TYPE "UDT_PECUpdateStatistics"
TITLE = UDT_PECupdateStatistics
VERSION : 0.1
//User-defined structure of FB_PECUpdate function block statistics.
   STRUCT
      PEC { S7_SetPoint := 'False'} : "UDT_PECStatistics";   // PEC Statistics
      TooManyLost { S7_SetPoint := 'False'} : "UDT_EventStatistic";   // Too many lost parcels
      TotalNrOfParcels : DInt;   // Total number of parcels
   END_STRUCT;

END_TYPE

TYPE "UDT_UnknownGIN"
TITLE = UDT_UnknownGIN
VERSION : 0.1
//User-defined structure of unknown GIN range.
   STRUCT
      Start : Int := 1;   // Unknown GIN range start value
      End : Int := 199;   // Unknown GIN range end value
      GIN : Int := 0;   // Las generated unknown GIN
   END_STRUCT;

END_TYPE

TYPE "UDT_AixPlcFullIn"
VERSION : 0.1
   STRUCT
      ConveyStopStatus { ExternalVisible := 'False'} : Struct   // Status of ConveyStop
         Bit08 { ExternalAccessible := 'False'; ExternalVisible := 'False'; ExternalWritable := 'False'} : Bool;   // Reserved
         Bit09 { ExternalAccessible := 'False'; ExternalVisible := 'False'; ExternalWritable := 'False'} : Bool;   // Reserved
         StopActiveCommandPLC { ExternalAccessible := 'False'; ExternalVisible := 'False'; ExternalWritable := 'False'} : Bool;   // Stop active due to stop command from the PLC
         Bit11 { ExternalAccessible := 'False'; ExternalVisible := 'False'; ExternalWritable := 'False'} : Bool;   // Reserved
         Bit12 { ExternalAccessible := 'False'; ExternalVisible := 'False'; ExternalWritable := 'False'} : Bool;   // Reserved
         Bit13 { ExternalAccessible := 'False'; ExternalVisible := 'False'; ExternalWritable := 'False'} : Bool;   // Reserved
         Bit14 { ExternalAccessible := 'False'; ExternalVisible := 'False'; ExternalWritable := 'False'} : Bool;   // Reserved
         Bit15 { ExternalAccessible := 'False'; ExternalVisible := 'False'; ExternalWritable := 'False'} : Bool;   // Reserved
         Bit00 { ExternalAccessible := 'False'; ExternalVisible := 'False'; ExternalWritable := 'False'} : Bool;   // Reserved
         Bit01 { ExternalAccessible := 'False'; ExternalVisible := 'False'; ExternalWritable := 'False'} : Bool;   // Reserved
         Bit02 { ExternalAccessible := 'False'; ExternalVisible := 'False'; ExternalWritable := 'False'} : Bool;   // Reserved
         Bit03 { ExternalAccessible := 'False'; ExternalVisible := 'False'; ExternalWritable := 'False'} : Bool;   // Reserved
         Bit04 { ExternalAccessible := 'False'; ExternalVisible := 'False'; ExternalWritable := 'False'} : Bool;   // Reserved
         StopActiveOtherModule { ExternalAccessible := 'False'; ExternalVisible := 'False'; ExternalWritable := 'False'} : Bool;   // Stop condition is active on a module in the ConveyStop group
         StopActiveLostConn { ExternalAccessible := 'False'; ExternalVisible := 'False'; ExternalWritable := 'False'} : Bool;   // Stop is active due to a loss of communication connection
         StopActiveLostPLC { ExternalAccessible := 'False'; ExternalVisible := 'False'; ExternalWritable := 'False'} : Bool;   // Stop active due to a loss of connection with the PLC
      END_STRUCT;
      AllSensorPortInputs { ExternalVisible := 'False'} : Struct   // Left and Right Sensor Port inputs
         Bit08 { ExternalAccessible := 'False'; ExternalVisible := 'False'; ExternalWritable := 'False'} : Bool;   // Reserved
         Bit09 { ExternalAccessible := 'False'; ExternalVisible := 'False'; ExternalWritable := 'False'} : Bool;   // Reserved
         Bit10 { ExternalAccessible := 'False'; ExternalVisible := 'False'; ExternalWritable := 'False'} : Bool;   // Reserved
         Bit11 { ExternalAccessible := 'False'; ExternalVisible := 'False'; ExternalWritable := 'False'} : Bool;   // Reserved
         Bit12 { ExternalAccessible := 'False'; ExternalVisible := 'False'; ExternalWritable := 'False'} : Bool;   // Reserved
         Bit13 { ExternalAccessible := 'False'; ExternalVisible := 'False'; ExternalWritable := 'False'} : Bool;   // Reserved
         Bit14 { ExternalAccessible := 'False'; ExternalVisible := 'False'; ExternalWritable := 'False'} : Bool;   // Reserved
         Heartbeat { ExternalAccessible := 'False'; ExternalVisible := 'False'; ExternalWritable := 'False'} : Bool;   // This bit toggles every 2 seconds
         LeftPin2 { ExternalAccessible := 'False'; ExternalVisible := 'False'; ExternalWritable := 'False'} : Bool;   // Left sensor port Pin2 state
         Bit01 { ExternalAccessible := 'False'; ExternalVisible := 'False'; ExternalWritable := 'False'} : Bool;   // Reserved
         RightPin2 { ExternalAccessible := 'False'; ExternalVisible := 'False'; ExternalWritable := 'False'} : Bool;   // Right sensor port Pin2 state
         Bit03 { ExternalAccessible := 'False'; ExternalVisible := 'False'; ExternalWritable := 'False'} : Bool;   // Reserved
         LeftSensor { ExternalAccessible := 'False'; ExternalVisible := 'False'; ExternalWritable := 'False'} : Bool;   // Left sensor port Pin4 state
         Bit05 { ExternalAccessible := 'False'; ExternalVisible := 'False'; ExternalWritable := 'False'} : Bool;   // Reserved
         RightSensor { ExternalAccessible := 'False'; ExternalVisible := 'False'; ExternalWritable := 'False'} : Bool;   // Right sensor port Pin4 state
         Bit07 { ExternalAccessible := 'False'; ExternalVisible := 'False'; ExternalWritable := 'False'} : Bool;   // Reserved
      END_STRUCT;
      SensorDetect { ExternalVisible := 'False'} : Struct   // Sensor detection
         Bits08_15 { ExternalVisible := 'False'} : SInt;   // Reserved
         RightSensorDetect { ExternalAccessible := 'False'; ExternalVisible := 'False'; ExternalWritable := 'False'} : Bool;   // True when sensor is detected
         LeftSensorDetect { ExternalAccessible := 'False'; ExternalVisible := 'False'; ExternalWritable := 'False'} : Bool;   // True when sensor is detected
         Bit02 { ExternalAccessible := 'False'; ExternalVisible := 'False'; ExternalWritable := 'False'} : Bool;   // Reserved
         Bit03 { ExternalAccessible := 'False'; ExternalVisible := 'False'; ExternalWritable := 'False'} : Bool;   // Reserved
         Bit04 { ExternalAccessible := 'False'; ExternalVisible := 'False'; ExternalWritable := 'False'} : Bool;   // Reserved
         Bit05 { ExternalAccessible := 'False'; ExternalVisible := 'False'; ExternalWritable := 'False'} : Bool;   // Reserved
         Bit06 { ExternalAccessible := 'False'; ExternalVisible := 'False'; ExternalWritable := 'False'} : Bool;   // Reserved
         Bit07 { ExternalAccessible := 'False'; ExternalVisible := 'False'; ExternalWritable := 'False'} : Bool;   // Reserved
      END_STRUCT;
      VoltageMotors { ExternalVisible := 'False'} : Int;   // The Voltage applied to the module's motor power connection in millivolts
      LeftMotorCurrent { ExternalVisible := 'False'} : Int;   // Left motor running current in milliamperes
      LeftMotorFreq { ExternalVisible := 'False'} : Int;   // Left motor running electrical frequency in Hz
      LeftMotorCalcTemp { ExternalVisible := 'False'} : Byte;   // Left motor temperature in degrees C
      ModuleTemp { ExternalVisible := 'False'} : Byte;   // Module CPU temperature in degrees C
      LeftMotorDiagnostic { ExternalVisible := 'False'} : Struct   // Left motor diagnostics .
         Overheat { ExternalAccessible := 'False'; ExternalVisible := 'False'; ExternalWritable := 'False'} : Bool;   // Left motor temperature has exceeded 105 degrees Celsius
         MaxTorque { ExternalAccessible := 'False'; ExternalVisible := 'False'; ExternalWritable := 'False'} : Bool;   // Left motor at maximum torque output
         ShortCircuit { ExternalAccessible := 'False'; ExternalVisible := 'False'; ExternalWritable := 'False'} : Bool;   // Left motor short circuit
         MotorNotConnected { ExternalAccessible := 'False'; ExternalVisible := 'False'; ExternalWritable := 'False'} : Bool;   // Left motor is not connected
         Overload { ExternalAccessible := 'False'; ExternalVisible := 'False'; ExternalWritable := 'False'} : Bool;   // Left motor overloaded after more than 20 seconds in Stalled
         Stalled { ExternalAccessible := 'False'; ExternalVisible := 'False'; ExternalWritable := 'False'} : Bool;   // Left motor stalled and speed is less than 10% of the set speed
         BadHall { ExternalAccessible := 'False'; ExternalVisible := 'False'; ExternalWritable := 'False'} : Bool;   // Left motor Hall Effect Sensor error active
         MotorNotUsed { ExternalAccessible := 'False'; ExternalVisible := 'False'; ExternalWritable := 'False'} : Bool;   // Left motor not used
         MotorStatus1 { ExternalAccessible := 'False'; ExternalVisible := 'False'; ExternalWritable := 'False'} : Bool;   // Left motor running and direction status
         MotorStatus2 { ExternalAccessible := 'False'; ExternalVisible := 'False'; ExternalWritable := 'False'} : Bool;   // Left motor running and direction status
         MotorPortinDOmode { ExternalAccessible := 'False'; ExternalVisible := 'False'; ExternalWritable := 'False'} : Bool;   // Left motor port is in digital Output mode .
         ReservedBit03 { ExternalAccessible := 'False'; ExternalVisible := 'False'; ExternalWritable := 'False'} : Bool;   // Reserved
         ReservedBit04 { ExternalAccessible := 'False'; ExternalVisible := 'False'; ExternalWritable := 'False'} : Bool;   // Reserved
         BoardOverheat { ExternalAccessible := 'False'; ExternalVisible := 'False'; ExternalWritable := 'False'} : Bool;   // Board temperature has exceeded 90 degrees Celsius
         OverVoltage { ExternalAccessible := 'False'; ExternalVisible := 'False'; ExternalWritable := 'False'} : Bool;   // Supply voltage + motor back EMF exceeded 30 volts
         LowVoltage { ExternalAccessible := 'False'; ExternalVisible := 'False'; ExternalWritable := 'False'} : Bool;   // Module power supply is less than 18 Volts
      END_STRUCT;
      RightMotorCurrent { ExternalVisible := 'False'} : Int;   // Right motor running current in milliamperes
      RightMotorFreq { ExternalVisible := 'False'} : Int;   // Right motor running electrical frequency in Hz
      RightMotorCalcTemp { ExternalVisible := 'False'} : Byte;   // Right motor temperature in degrees Celsius
      ModuleTemp1 { ExternalVisible := 'False'} : Byte;   // Module PCB temperature in degrees C (same as ModuleTemp tag)
      RightMotorDiagnostic { ExternalVisible := 'False'} : Struct   // Right motor diagnostics .
         Overheat { ExternalAccessible := 'False'; ExternalVisible := 'False'; ExternalWritable := 'False'} : Bool;   // Right motor temperature has exceeded 105 degrees Celsius
         MaxTorque { ExternalAccessible := 'False'; ExternalVisible := 'False'; ExternalWritable := 'False'} : Bool;   // Right motor at maximum torque output
         ShortCircuit { ExternalAccessible := 'False'; ExternalVisible := 'False'; ExternalWritable := 'False'} : Bool;   // Right motor short circuit
         MotorNotConnected { ExternalAccessible := 'False'; ExternalVisible := 'False'; ExternalWritable := 'False'} : Bool;   // Right motor is not connected
         Overload { ExternalAccessible := 'False'; ExternalVisible := 'False'; ExternalWritable := 'False'} : Bool;   // Right motor overloaded after more than 20 seconds in Stalled
         Stalled { ExternalAccessible := 'False'; ExternalVisible := 'False'; ExternalWritable := 'False'} : Bool;   // Right motor stalled and speed is less than 10% of the set speed
         BadHall { ExternalAccessible := 'False'; ExternalVisible := 'False'; ExternalWritable := 'False'} : Bool;   // Right motor Hall Effect Sensor error active
         MotorNotUsed { ExternalAccessible := 'False'; ExternalVisible := 'False'; ExternalWritable := 'False'} : Bool;   // Right motor is not used
         MotorStatus1 { ExternalAccessible := 'False'; ExternalVisible := 'False'; ExternalWritable := 'False'} : Bool;   // Right motor running and direction status
         MotorStatus2 { ExternalAccessible := 'False'; ExternalVisible := 'False'; ExternalWritable := 'False'} : Bool;   // Right motor running and direction status
         MotorPortinDOmode { ExternalAccessible := 'False'; ExternalVisible := 'False'; ExternalWritable := 'False'} : Bool;   // Right motor port is in digital output mode .
         ReservedBit03 { ExternalAccessible := 'False'; ExternalVisible := 'False'; ExternalWritable := 'False'} : Bool;   // Reserved
         ReservedBit04 { ExternalAccessible := 'False'; ExternalVisible := 'False'; ExternalWritable := 'False'} : Bool;   // Reserved
         BoardOverheat { ExternalAccessible := 'False'; ExternalVisible := 'False'; ExternalWritable := 'False'} : Bool;   // Board temperature has exceeded 90 degrees Celsius
         OverVoltage { ExternalAccessible := 'False'; ExternalVisible := 'False'; ExternalWritable := 'False'} : Bool;   // Supply voltage + motor back EMF exceeded 30 volts
         LowVoltage { ExternalAccessible := 'False'; ExternalVisible := 'False'; ExternalWritable := 'False'} : Bool;   // Module power supply is less than 18 Volts
      END_STRUCT;
      LeftMotorDIOstatus { ExternalVisible := 'False'} : Struct   // Status of Left M8 motor port when used as a digital IO
         Bit08 { ExternalAccessible := 'False'; ExternalVisible := 'False'; ExternalWritable := 'False'} : Bool;   // Reserved
         Bit09 { ExternalAccessible := 'False'; ExternalVisible := 'False'; ExternalWritable := 'False'} : Bool;   // Reserved
         Bit10 { ExternalAccessible := 'False'; ExternalVisible := 'False'; ExternalWritable := 'False'} : Bool;   // Reserved
         Bit11 { ExternalAccessible := 'False'; ExternalVisible := 'False'; ExternalWritable := 'False'} : Bool;   // Reserved
         ShortCircuit { ExternalAccessible := 'False'; ExternalVisible := 'False'; ExternalWritable := 'False'} : Bool;   // Short circuit between +24V and any of the U,V,W phases
         Bit13 { ExternalAccessible := 'False'; ExternalVisible := 'False'; ExternalWritable := 'False'} : Bool;   // Reserved
         Bit14 { ExternalAccessible := 'False'; ExternalVisible := 'False'; ExternalWritable := 'False'} : Bool;   // Reserved
         Bit15 { ExternalAccessible := 'False'; ExternalVisible := 'False'; ExternalWritable := 'False'} : Bool;   // Reserved
         Bits00_07 { ExternalVisible := 'False'} : SInt;   // Reserved
      END_STRUCT;
      RightMotorDIOstatus { ExternalVisible := 'False'} : Struct   // Status of Right M8 motor port when used as a digital IO
         Bit08 { ExternalAccessible := 'False'; ExternalVisible := 'False'; ExternalWritable := 'False'} : Bool;   // Reserved
         Bit09 { ExternalAccessible := 'False'; ExternalVisible := 'False'; ExternalWritable := 'False'} : Bool;   // Reserved
         Bit10 { ExternalAccessible := 'False'; ExternalVisible := 'False'; ExternalWritable := 'False'} : Bool;   // Reserved
         Bit11 { ExternalAccessible := 'False'; ExternalVisible := 'False'; ExternalWritable := 'False'} : Bool;   // Reserved
         ShortCircuit { ExternalAccessible := 'False'; ExternalVisible := 'False'; ExternalWritable := 'False'} : Bool;   // Short circuit between +24V and any of the U,V,W phases
         Bit13 { ExternalAccessible := 'False'; ExternalVisible := 'False'; ExternalWritable := 'False'} : Bool;   // Reserved
         Bit14 { ExternalAccessible := 'False'; ExternalVisible := 'False'; ExternalWritable := 'False'} : Bool;   // Reserved
         Bit15 { ExternalAccessible := 'False'; ExternalVisible := 'False'; ExternalWritable := 'False'} : Bool;   // Reserved
         Bits00_07 { ExternalVisible := 'False'} : SInt;   // Reserved
      END_STRUCT;
      UpstreamModuleStatus { ExternalVisible := 'False'} : Word;   // The ZPA status from the Upstream ConveyLinx module
      DownstreamModuleStatus { ExternalVisible := 'False'} : Word;   // The ZPA status from the Downstream ConveyLinx module
      TrackingFromUpstream { ExternalVisible := 'False'} : DWord;   // Tracking data from the Upstream ConveyLinx module
      Index18 { ExternalVisible := 'False'} : Word;   // Index
      ServoLocationLeft { ExternalVisible := 'False'} : Int;   // Left motor current location from 0 in mm for MDR and in pulses for PGD
      ServoLocationRight { ExternalVisible := 'False'} : Int;   // Right motor current location from 0 in mm for MDR and in pulses for PGD
      ServoStatusLeft { ExternalVisible := 'False'} : Word;   // Left motor servo commands status
      ServoStatusRight { ExternalVisible := 'False'} : Word;   // Right motor servo commands status
      LeftMotorActualSpeed { ExternalVisible := 'False'} : Word;   // Bits 0 thru 13: Left motor actual speed in mm/sec, Bits 14-15: Status. For PGD, base unit is 1/10 RPM
      RightMotorActualSpeed { ExternalVisible := 'False'} : Word;   // Bits 0 thru 13: Left motor actual speed in mm/sec, Bits 14-15: Status. For PGD, base unit is 1/10 RPM
      Future { ExternalVisible := 'False'} : Array[25..31] of Int;   // Future
   END_STRUCT;

END_TYPE

TYPE "UDT_AixPlcFullOut"
VERSION : 0.1
   STRUCT
      ConveyStopControl { ExternalVisible := 'False'} : Word;   // Writing '1' causes the Stop group to go into STOP state . Transition 0 - 2 is needed to clear the Stop
      LeftMotorAsDIO { ExternalVisible := 'False'} : Struct   // Use the Left M8 motor port as digital IO
         Bit08 { ExternalAccessible := 'False'; ExternalVisible := 'False'; ExternalWritable := 'False'} : Bool;   // Reserved
         Bit09 { ExternalAccessible := 'False'; ExternalVisible := 'False'; ExternalWritable := 'False'} : Bool;   // Reserved
         Bit10 { ExternalAccessible := 'False'; ExternalVisible := 'False'; ExternalWritable := 'False'} : Bool;   // Reserved
         Bit11 { ExternalAccessible := 'False'; ExternalVisible := 'False'; ExternalWritable := 'False'} : Bool;   // Reserved
         Bit12 { ExternalAccessible := 'False'; ExternalVisible := 'False'; ExternalWritable := 'False'} : Bool;   // Reserved
         Bit13 { ExternalAccessible := 'False'; ExternalVisible := 'False'; ExternalWritable := 'False'} : Bool;   // Reserved
         Bit14 { ExternalAccessible := 'False'; ExternalVisible := 'False'; ExternalWritable := 'False'} : Bool;   // Reserved
         EnableDIO { ExternalAccessible := 'False'; ExternalVisible := 'False'; ExternalWritable := 'False'} : Bool;   // Set bit to enable Left motor M8 port Digital IO mode
         Bit00 { ExternalAccessible := 'False'; ExternalVisible := 'False'; ExternalWritable := 'False'} : Bool;   // Reserved
         EnergizeM8Pin4 { ExternalAccessible := 'False'; ExternalVisible := 'False'; ExternalWritable := 'False'} : Bool;   // Energize motor port M8 PIN 4
         EnergizeM8Pin3 { ExternalAccessible := 'False'; ExternalVisible := 'False'; ExternalWritable := 'False'} : Bool;   // Energize motor port M8 PIN 3
         Bit03 { ExternalAccessible := 'False'; ExternalVisible := 'False'; ExternalWritable := 'False'} : Bool;   // Reserved
         Bit04 { ExternalAccessible := 'False'; ExternalVisible := 'False'; ExternalWritable := 'False'} : Bool;   // Reserved
         Bit05 { ExternalAccessible := 'False'; ExternalVisible := 'False'; ExternalWritable := 'False'} : Bool;   // Reserved
         Bit06 { ExternalAccessible := 'False'; ExternalVisible := 'False'; ExternalWritable := 'False'} : Bool;   // Reserved
         Bit07 { ExternalAccessible := 'False'; ExternalVisible := 'False'; ExternalWritable := 'False'} : Bool;   // Reserved
      END_STRUCT;
      RightMotorAsDIO { ExternalVisible := 'False'} : Struct   // Use the Right M8 motor port as digital IO
         Bit08 { ExternalAccessible := 'False'; ExternalVisible := 'False'; ExternalWritable := 'False'} : Bool;   // Reserved
         Bit09 { ExternalAccessible := 'False'; ExternalVisible := 'False'; ExternalWritable := 'False'} : Bool;   // Reserved
         Bit10 { ExternalAccessible := 'False'; ExternalVisible := 'False'; ExternalWritable := 'False'} : Bool;   // Reserved
         Bit11 { ExternalAccessible := 'False'; ExternalVisible := 'False'; ExternalWritable := 'False'} : Bool;   // Reserved
         Bit12 { ExternalAccessible := 'False'; ExternalVisible := 'False'; ExternalWritable := 'False'} : Bool;   // Reserved
         Bit13 { ExternalAccessible := 'False'; ExternalVisible := 'False'; ExternalWritable := 'False'} : Bool;   // Reserved
         Bit14 { ExternalAccessible := 'False'; ExternalVisible := 'False'; ExternalWritable := 'False'} : Bool;   // Reserved
         EnableDIO { ExternalAccessible := 'False'; ExternalVisible := 'False'; ExternalWritable := 'False'} : Bool;   // Set bit to enable Left motor M8 port Digital IO mode
         EnergizeM8Pin2 { ExternalAccessible := 'False'; ExternalVisible := 'False'; ExternalWritable := 'False'} : Bool;   // Energize motor port M8 PIN 2
         Bit01 { ExternalAccessible := 'False'; ExternalVisible := 'False'; ExternalWritable := 'False'} : Bool;   // Reserved
         EnergizeM8Pin3 { ExternalAccessible := 'False'; ExternalVisible := 'False'; ExternalWritable := 'False'} : Bool;   // Energize motor port M8 PIN 3
         Bit03 { ExternalAccessible := 'False'; ExternalVisible := 'False'; ExternalWritable := 'False'} : Bool;   // Reserved
         Bit04 { ExternalAccessible := 'False'; ExternalVisible := 'False'; ExternalWritable := 'False'} : Bool;   // Reserved
         Bit05 { ExternalAccessible := 'False'; ExternalVisible := 'False'; ExternalWritable := 'False'} : Bool;   // Reserved
         Bit06 { ExternalAccessible := 'False'; ExternalVisible := 'False'; ExternalWritable := 'False'} : Bool;   // Reserved
         Bit07 { ExternalAccessible := 'False'; ExternalVisible := 'False'; ExternalWritable := 'False'} : Bool;   // Reserved
      END_STRUCT;
      SensorPortsDO { ExternalVisible := 'False'} : Struct   // The Sensor ports PIN2 as digital outputs
         Bit08 { ExternalAccessible := 'False'; ExternalVisible := 'False'; ExternalWritable := 'False'} : Bool;   // Reserved
         Bit09 { ExternalAccessible := 'False'; ExternalVisible := 'False'; ExternalWritable := 'False'} : Bool;   // Reserved
         Bit10 { ExternalAccessible := 'False'; ExternalVisible := 'False'; ExternalWritable := 'False'} : Bool;   // Reserved
         Bit11 { ExternalAccessible := 'False'; ExternalVisible := 'False'; ExternalWritable := 'False'} : Bool;   // Reserved
         Bit12 { ExternalAccessible := 'False'; ExternalVisible := 'False'; ExternalWritable := 'False'} : Bool;   // Reserved
         Bit13 { ExternalAccessible := 'False'; ExternalVisible := 'False'; ExternalWritable := 'False'} : Bool;   // Reserved
         Bit14 { ExternalAccessible := 'False'; ExternalVisible := 'False'; ExternalWritable := 'False'} : Bool;   // Reserved
         Bit15 { ExternalAccessible := 'False'; ExternalVisible := 'False'; ExternalWritable := 'False'} : Bool;   // Reserved
         EnergizeLeftPortPin2 { ExternalAccessible := 'False'; ExternalVisible := 'False'; ExternalWritable := 'False'} : Bool;   // Set to turn on Left Port Pin2
         EnergizeRightPortPin2 { ExternalAccessible := 'False'; ExternalVisible := 'False'; ExternalWritable := 'False'} : Bool;   // Set to turn on Right Port Pin2
         Bit02 { ExternalAccessible := 'False'; ExternalVisible := 'False'; ExternalWritable := 'False'} : Bool;   // Reserved
         Bit03 { ExternalAccessible := 'False'; ExternalVisible := 'False'; ExternalWritable := 'False'} : Bool;   // Reserved
         Bit04 { ExternalAccessible := 'False'; ExternalVisible := 'False'; ExternalWritable := 'False'} : Bool;   // Reserved
         EnableLeftPortPin2 { ExternalAccessible := 'False'; ExternalVisible := 'False'; ExternalWritable := 'False'} : Bool;   // Set to enable, reset for Pin2  to be input
         EnableRightPortPin2 { ExternalAccessible := 'False'; ExternalVisible := 'False'; ExternalWritable := 'False'} : Bool;   // Set to enable, reset for Pin2  to be input
         Bit07 { ExternalAccessible := 'False'; ExternalVisible := 'False'; ExternalWritable := 'False'} : Bool;   // Reserved
      END_STRUCT;
      LeftMotorControl { ExternalVisible := 'False'} : Struct   // Run/Stop and Direction control of the Left motor
         MotorDirection { ExternalAccessible := 'False'; ExternalVisible := 'False'; ExternalWritable := 'False'} : Bool;   // 0 = Configured direction /1 = opposite to configured direction
         Bit09 { ExternalAccessible := 'False'; ExternalVisible := 'False'; ExternalWritable := 'False'} : Bool;   // Reserved
         Bit10 { ExternalAccessible := 'False'; ExternalVisible := 'False'; ExternalWritable := 'False'} : Bool;   // Reserved
         Bit11 { ExternalAccessible := 'False'; ExternalVisible := 'False'; ExternalWritable := 'False'} : Bool;   // Reserved
         Bit12 { ExternalAccessible := 'False'; ExternalVisible := 'False'; ExternalWritable := 'False'} : Bool;   // Reserved
         Bit13 { ExternalAccessible := 'False'; ExternalVisible := 'False'; ExternalWritable := 'False'} : Bool;   // Reserved
         Bit14 { ExternalAccessible := 'False'; ExternalVisible := 'False'; ExternalWritable := 'False'} : Bool;   // Reserved
         Bit15 { ExternalAccessible := 'False'; ExternalVisible := 'False'; ExternalWritable := 'False'} : Bool;   // Reserved
         Run { ExternalAccessible := 'False'; ExternalVisible := 'False'; ExternalWritable := 'False'} : Bool;   // Run = 1 / Stop = 0
         Bit01 { ExternalAccessible := 'False'; ExternalVisible := 'False'; ExternalWritable := 'False'} : Bool;   // Reserved
         Bit02 { ExternalAccessible := 'False'; ExternalVisible := 'False'; ExternalWritable := 'False'} : Bool;   // Reserved
         Bit03 { ExternalAccessible := 'False'; ExternalVisible := 'False'; ExternalWritable := 'False'} : Bool;   // Reserved
         Bit04 { ExternalAccessible := 'False'; ExternalVisible := 'False'; ExternalWritable := 'False'} : Bool;   // Reserved
         Bit05 { ExternalAccessible := 'False'; ExternalVisible := 'False'; ExternalWritable := 'False'} : Bool;   // Reserved
         Bit06 { ExternalAccessible := 'False'; ExternalVisible := 'False'; ExternalWritable := 'False'} : Bool;   // Reserved
         Bit07 { ExternalAccessible := 'False'; ExternalVisible := 'False'; ExternalWritable := 'False'} : Bool;   // Reserved
      END_STRUCT;
      LeftSetMotorBrakeMode { ExternalVisible := 'False'} : Word;   // Set Left motor Brake Mode.0 = ignore 1 = "Normal" / 2 = "Free" / 3 ="Servo brake"
      LeftSetMotorSlaveMode { ExternalVisible := 'False'} : Word;   // 0 = ignore  1=Off, Left Independant  2=On, Left Mirror Right   3=On, Left Opposite Right direction
      RightMotorControl { ExternalVisible := 'False'} : Struct   // Run/Stop and Direction control of the Right motor
         MotorDirection { ExternalAccessible := 'False'; ExternalVisible := 'False'; ExternalWritable := 'False'} : Bool;   // 0 = Configured direction /1 = opposite to configured direction
         Bit09 { ExternalAccessible := 'False'; ExternalVisible := 'False'; ExternalWritable := 'False'} : Bool;   // Reserved
         Bit10 { ExternalAccessible := 'False'; ExternalVisible := 'False'; ExternalWritable := 'False'} : Bool;   // Reserved
         Bit11 { ExternalAccessible := 'False'; ExternalVisible := 'False'; ExternalWritable := 'False'} : Bool;   // Reserved
         Bit12 { ExternalAccessible := 'False'; ExternalVisible := 'False'; ExternalWritable := 'False'} : Bool;   // Reserved
         Bit13 { ExternalAccessible := 'False'; ExternalVisible := 'False'; ExternalWritable := 'False'} : Bool;   // Reserved
         Bit14 { ExternalAccessible := 'False'; ExternalVisible := 'False'; ExternalWritable := 'False'} : Bool;   // Reserved
         Bit15 { ExternalAccessible := 'False'; ExternalVisible := 'False'; ExternalWritable := 'False'} : Bool;   // Reserved
         Run { ExternalAccessible := 'False'; ExternalVisible := 'False'; ExternalWritable := 'False'} : Bool;   // Run = 1 / Stop = 0
         Bit01 { ExternalAccessible := 'False'; ExternalVisible := 'False'; ExternalWritable := 'False'} : Bool;   // Reserved
         Bit02 { ExternalAccessible := 'False'; ExternalVisible := 'False'; ExternalWritable := 'False'} : Bool;   // Reserved
         Bit03 { ExternalAccessible := 'False'; ExternalVisible := 'False'; ExternalWritable := 'False'} : Bool;   // Reserved
         Bit04 { ExternalAccessible := 'False'; ExternalVisible := 'False'; ExternalWritable := 'False'} : Bool;   // Reserved
         Bit05 { ExternalAccessible := 'False'; ExternalVisible := 'False'; ExternalWritable := 'False'} : Bool;   // Reserved
         Bit06 { ExternalAccessible := 'False'; ExternalVisible := 'False'; ExternalWritable := 'False'} : Bool;   // Reserved
         Bit07 { ExternalAccessible := 'False'; ExternalVisible := 'False'; ExternalWritable := 'False'} : Bool;   // Reserved
      END_STRUCT;
      RightSetMotorBrakeMode { ExternalVisible := 'False'} : Word;   // Set Right motor Brake Mode.0 = ignore 1 = "Normal" / 2 = "Free" / 3 ="Servo brake"
      RightSetMotorSlaveMode { ExternalVisible := 'False'} : Word;   // 0 = ignore 1=Off, Right Independant  2=On, Right Mirror Right   3=On, Right Opposite Right direction
      LeftSetMotorSpeed { ExternalVisible := 'False'} : Int;   // Set reference speed for Left motor in mm/s (or 1/10 of an RPM for PGD)
      RightSetMotorSpeed { ExternalVisible := 'False'} : Int;   // Set reference speed for Right motor mm/s  (or 1/10 of an RPM for PGD)
      LeftSetMotorAccel { ExternalVisible := 'False'} : Int;   // Set acceleration distance in mm for Left motor (or pulses for PGD)
      LeftSetMotorDeccel { ExternalVisible := 'False'} : Int;   // Set deceleration distance in mm for Left motor (or pulses for PGD)
      RightSetMotorAccel { ExternalVisible := 'False'} : Int;   // Set acceleration distance in mm for Right motor (or pulses for PGD)
      RightSetMotorDeccel { ExternalVisible := 'False'} : Int;   // Set deceleration distance in mm for Right motor (or pulses for PGD)
      ClearMotorError { ExternalVisible := 'False'} : Word;   // Write '1' to clear motor error, wait 500 msec, then write '0' return to operation
      SendStatusToDownstream { ExternalVisible := 'False'} : Word;   // Write '4' or '5' to signal downstream ConveyLinx module in ZPA mode to wake up
      SendStatusToUpstream { ExternalVisible := 'False'} : Word;   // Write '5' to signal upstream ConveyLinx module in ZPA mode to accumulate, write '1' to signal OK to receive
      SensorPolarity { ExternalVisible := 'False'} : Struct   // Set logic polarity for Sensor Port's PIN2 and PIN4
         Bit08 { ExternalAccessible := 'False'; ExternalVisible := 'False'; ExternalWritable := 'False'} : Bool;   // Reserved
         Bit09 { ExternalAccessible := 'False'; ExternalVisible := 'False'; ExternalWritable := 'False'} : Bool;   // Reserved
         Bit10 { ExternalAccessible := 'False'; ExternalVisible := 'False'; ExternalWritable := 'False'} : Bool;   // Reserved
         Bit11 { ExternalAccessible := 'False'; ExternalVisible := 'False'; ExternalWritable := 'False'} : Bool;   // Reserved
         Bit12 { ExternalAccessible := 'False'; ExternalVisible := 'False'; ExternalWritable := 'False'} : Bool;   // Reserved
         Bit13 { ExternalAccessible := 'False'; ExternalVisible := 'False'; ExternalWritable := 'False'} : Bool;   // Reserved
         Bit14 { ExternalAccessible := 'False'; ExternalVisible := 'False'; ExternalWritable := 'False'} : Bool;   // Reserved
         Bit15 { ExternalAccessible := 'False'; ExternalVisible := 'False'; ExternalWritable := 'False'} : Bool;   // Reserved
         Left_Pin2 { ExternalAccessible := 'False'; ExternalVisible := 'False'; ExternalWritable := 'False'} : Bool;   // Set to invert, reset for normal
         Bit01 { ExternalAccessible := 'False'; ExternalVisible := 'False'; ExternalWritable := 'False'} : Bool;   // Reserved
         Right_Pin2 { ExternalAccessible := 'False'; ExternalVisible := 'False'; ExternalWritable := 'False'} : Bool;   // Set to invert, reset for normal
         Bit03 { ExternalAccessible := 'False'; ExternalVisible := 'False'; ExternalWritable := 'False'} : Bool;   // Reserved
         Left_Pin4 { ExternalAccessible := 'False'; ExternalVisible := 'False'; ExternalWritable := 'False'} : Bool;   // Set to invert, reset for normal
         Bit05 { ExternalAccessible := 'False'; ExternalVisible := 'False'; ExternalWritable := 'False'} : Bool;   // Reserved
         Right_Pin4 { ExternalAccessible := 'False'; ExternalVisible := 'False'; ExternalWritable := 'False'} : Bool;   // Set to invert, reset for normal
         Bit07 { ExternalAccessible := 'False'; ExternalVisible := 'False'; ExternalWritable := 'False'} : Bool;   // Reserved
      END_STRUCT;
      TrackingToDownstream { ExternalVisible := 'False'} : DWord;   // Write Tracking data to be captured by downstream ZPA mode ConveyLinx
      Index22 { ExternalVisible := 'False'} : Word;   // Reserved
      ServoControlDistanceLeft { ExternalVisible := 'False'} : Int;   // Position from 0 in mm for Left motor to move on next command
      ServoControlCommandLeft { ExternalVisible := 'False'} : Word;   // Left motor servo command
      ServoControlDistanceRight { ExternalVisible := 'False'} : Int;   // New position from 0 in mm for Right motor to move on next command
      ServoControlCommandRight { ExternalVisible := 'False'} : Word;   // Right motor servo command
      Future { ExternalVisible := 'False'} : Array[27..31] of Int;   // Reserved
   END_STRUCT;

END_TYPE

TYPE "UDT_PECUpdateStatus"
TITLE = UDT_PECUpdateStatus
VERSION : 0.1
//User-defined structure of FB_PECUpdate function block status.
   STRUCT
      TooManyLost { ExternalAccessible := 'False'; ExternalVisible := 'False'; ExternalWritable := 'False'} : Bool;   // Too many parcels lost in a row
      LowPerformance { ExternalAccessible := 'False'; ExternalVisible := 'False'; ExternalWritable := 'False'} : Bool;   // Performance warning
      PEC { ExternalAccessible := 'False'; ExternalVisible := 'False'; ExternalWritable := 'False'} : Bool;   // Current state of the end of section photo eye
      Jam { ExternalAccessible := 'False'; ExternalVisible := 'False'; ExternalWritable := 'False'} : Bool;   // PEC Jam error
   END_STRUCT;

END_TYPE

FUNCTION_BLOCK "FB_Pulse"
TITLE = FB_Pulse
{ S7_Optimized_Access := 'TRUE' }
AUTHOR : MHSE
FAMILY : GeneralSystemFunctions
VERSION : 3.0
// ATTRIBUTES
// AUTO_NUMBER = True
// BLOCK_NUMBER = 26
// END_ATTRIBUTES
//Function block to generate custom pulse signal.
   VAR_INPUT
      iudi_PulseTime { ExternalAccessible := 'False'; ExternalVisible := 'False'; ExternalWritable := 'False'} : UDInt;   // Pulse time [ms]
   END_VAR

   VAR_OUTPUT
      qx_Pulse { ExternalAccessible := 'False'; ExternalVisible := 'False'; ExternalWritable := 'False'} : Bool;   // Pulse output
   END_VAR

   VAR
      R_TRIG {InstructionName := 'R_TRIG'; LibVersion := '1.0'; ExternalAccessible := 'False'; ExternalVisible := 'False'; ExternalWritable := 'False'; S7_SetPoint := 'False'} : R_TRIG;   // Siemens "R_Trig" - to prepare rising edge trigger on "sx_Pulse" signal
      slr_ActualPulseTime { ExternalAccessible := 'False'; ExternalVisible := 'False'; ExternalWritable := 'False'} : LReal;   // Actual pulse time [ms]
      sx_Pulse { ExternalAccessible := 'False'; ExternalVisible := 'False'; ExternalWritable := 'False'} : Bool;   // Pulse signal
   END_VAR


BEGIN
	(*
	----------------------------------------------------------------------------------------

	Version history:
	Date        | Version   | Author        | Remark
	----------------------------------------------------------------------------------------
	24/05/2019  | 0.1       | K.Pokorski    | first release MHS TIA 15.1
	24/07/2019  | 2.0       | L.Klar        | 2.0 MHS library release TIA 15.1
	27/08/2019  | 2.1       | K.Pokorski    | Comments adjusted
	04/11/2019  | 2.2       | L.Klar        | Prevoius cycle scan changed from memory to DB variable
	12/11/2019  | 3.0       | P.Majka       | 3.0 MHS library release TIA 15.1
	21/02/2023  | 4.0       | F.Baten       | 4.0 Release TIA 17.5
	*)

	REGION 1 - Pulse calculation

	    // Pulse timer on
	    IF (#iudi_PulseTime <= #slr_ActualPulseTime)
	    THEN

	        #sx_Pulse := TRUE;
	        #slr_ActualPulseTime := 0;

	    ELSE

	        #slr_ActualPulseTime += "DB_Memory".PrevCycleTime;
	        #sx_Pulse := FALSE;

	    END_IF;

	END_REGION

	REGION 2 - Pulse output

	    #R_TRIG(CLK := #sx_Pulse,
	            Q => #qx_Pulse);

	END_REGION
END_FUNCTION_BLOCK

FUNCTION "FC_BitAllocation" : Void
{ S7_Optimized_Access := 'TRUE' }
VERSION : 0.1
   VAR_INPUT
      ix_Bit0 : Bool;
      ix_Bit1 : Bool;
      ix_Bit2 : Bool;
      ix_Bit3 : Bool;
      ix_Bit4 : Bool;
      ix_Bit5 : Bool;
      ix_Bit6 : Bool;
      ix_Bit7 : Bool;
      ix_Bit8 : Bool;
      ix_Bit9 : Bool;
      ix_Bit10 : Bool;
      ix_Bit11 : Bool;
      ix_Bit12 : Bool;
      ix_Bit13 : Bool;
      ix_Bit14 : Bool;
      ix_Bit15 : Bool;
      ix_Bit16 : Bool;
      ix_Bit17 : Bool;
      ix_Bit18 : Bool;
      ix_Bit19 : Bool;
      ix_Bit20 : Bool;
      ix_Bit21 : Bool;
      ix_Bit22 : Bool;
      ix_Bit23 : Bool;
      ix_Bit24 : Bool;
      ix_Bit25 : Bool;
      ix_Bit26 : Bool;
      ix_Bit27 : Bool;
      ix_Bit28 : Bool;
      ix_Bit29 : Bool;
      ix_Bit30 : Bool;
      ix_Bit31 : Bool;
   END_VAR

   VAR_OUTPUT
      qdw_Dword : DWord;
   END_VAR


BEGIN
	#qdw_Dword.%X0 := #ix_Bit0;
	#qdw_Dword.%X1 := #ix_Bit1;
	#qdw_Dword.%X2 := #ix_Bit2;
	#qdw_Dword.%X3 := #ix_Bit3;
	#qdw_Dword.%X4 := #ix_Bit4;
	#qdw_Dword.%X5 := #ix_Bit5;
	#qdw_Dword.%X6 := #ix_Bit6;
	#qdw_Dword.%X7 := #ix_Bit7;
	#qdw_Dword.%X8 := #ix_Bit8;
	#qdw_Dword.%X9 := #ix_Bit9;
	#qdw_Dword.%X10 := #ix_Bit10;
	#qdw_Dword.%X11 := #ix_Bit11;
	#qdw_Dword.%X12 := #ix_Bit12;
	#qdw_Dword.%X13 := #ix_Bit13;
	#qdw_Dword.%X14 := #ix_Bit14;
	#qdw_Dword.%X15 := #ix_Bit15;
	#qdw_Dword.%X16 := #ix_Bit16;
	#qdw_Dword.%X17 := #ix_Bit17;
	#qdw_Dword.%X18 := #ix_Bit18;
	#qdw_Dword.%X19 := #ix_Bit19;
	#qdw_Dword.%X20 := #ix_Bit20;
	#qdw_Dword.%X21 := #ix_Bit21;
	#qdw_Dword.%X22 := #ix_Bit22;
	#qdw_Dword.%X23 := #ix_Bit23;
	#qdw_Dword.%X24 := #ix_Bit24;
	#qdw_Dword.%X25 := #ix_Bit25;
	#qdw_Dword.%X26 := #ix_Bit26;
	#qdw_Dword.%X27 := #ix_Bit27;
	#qdw_Dword.%X28 := #ix_Bit28;
	#qdw_Dword.%X29 := #ix_Bit29;
	#qdw_Dword.%X30 := #ix_Bit30;
	#qdw_Dword.%X31 := #ix_Bit31;

END_FUNCTION

TYPE "UDT_PECUpdateConfiguration"
TITLE = UDT_PECConfiguration
VERSION : 0.1
//User-defined structure of PEC parameters.
   STRUCT
      Distance : DInt;   // Distance between photo eye and the end of conveyor [mm]
      JamDisplacementLimit : Int;   // Limit displacement with PEC blocked o detect jam [cm]
      TimeOnDelay : UDInt;   // Photo eye time on delay [ms]
      TimeOffDelay : UDInt;   // Photo eye time off delay [ms]
      ParcelLengthFilter : Bool := TRUE;   // Parcel length filter
      ResetWithPECBlocked { ExternalAccessible := 'False'; ExternalVisible := 'False'; ExternalWritable := 'False'} : Bool;   // When 'True' Allow reset system after jam with PEC blocked
      SearchWindowFwd : Int;   // Search window in forward direction [cm]
      SearchWindowRvs : Int;   // Search window in reverse direction [cm]
      GINRangeStart : Int;   // GIN range start value
      GINRangeEnd : Int;   // GIN range end value
      NrOfTeachParcels : Int;   // Number of parcels to teach
      DefaultGIN : Int := 1;   // Default GIN record
      MaxLost : Int;   // Maximum number of lost parcels in a row
      GenerationPoint { ExternalAccessible := 'False'; ExternalVisible := 'False'; ExternalWritable := 'False'} : Bool;   // Generation point
      NegativeGINDelete { ExternalAccessible := 'False'; ExternalVisible := 'False'; ExternalWritable := 'False'} : Bool;   // True when negative GIN has to be deleted
      ParcelLengthMeasurement { ExternalAccessible := 'False'; ExternalVisible := 'False'; ExternalWritable := 'False'} : Bool;   // Parcel length measurement
      GapLengthMeasurement { ExternalAccessible := 'False'; ExternalVisible := 'False'; ExternalWritable := 'False'} : Bool;   // Gap length measurement
   END_STRUCT;

END_TYPE

TYPE "UDT_ValveStatistics"
VERSION : 0.1
   STRUCT
      Open : "UDT_EventStatistic";   // Number of times PEC got jammed
      Fail : "UDT_EventStatistic";
   END_STRUCT;

END_TYPE

TYPE "UDT_PendantVT100Statistics"
VERSION : 0.1
   STRUCT
      PNSlaveError : "UDT_EventStatistic";   // Statistics of a Profinet slave error
      PNSlaveNotOnline : "UDT_EventStatistic";   // Statistics of  Profinet slave not online
   END_STRUCT;

END_TYPE

TYPE "UDT_LoaderStatistics"
TITLE = UDT_LoaderStatistics
VERSION : 0.1
//User-defined structure of FB_Loader function block statistics.
   STRUCT
      EnergySave : "UDT_EventStatistic";   // Number of times that save energy mode occurs
      ExtendableUpTime : "UDT_EventStatistic";   // Conveyor up time
      ExtendableDownTime : "UDT_EventStatistic";   // Conveyor down time
      VFDError : "UDT_EventStatistic";   // VFD Error
      NotHealthy : "UDT_EventStatistic";   // Extendable not healthy
   END_STRUCT;

END_TYPE

TYPE "UDT_LoaderStatus"
TITLE = UDT_LoaderStatus
VERSION : 0.1
//User-defined structure of FB_Loader function block status.
   STRUCT
      Status : Int;   // Status number
      Specific : Struct   // Equipment specific warnings and errors
         Disabled { ExternalAccessible := 'False'; ExternalVisible := 'False'; ExternalWritable := 'False'} : Bool;   // Loader is disabled by HMI
         VFDError { ExternalAccessible := 'False'; ExternalVisible := 'False'; ExternalWritable := 'False'} : Bool;   // Loader has an VFD error
         NotHealthy { ExternalAccessible := 'False'; ExternalVisible := 'False'; ExternalWritable := 'False'} : Bool;   // Loader is not healthy
         StoreMode { ExternalAccessible := 'False'; ExternalVisible := 'False'; ExternalWritable := 'False'} : Bool;   // Extendable is in store mode
         FeedMode { ExternalAccessible := 'False'; ExternalVisible := 'False'; ExternalWritable := 'False'} : Bool;   // Extendable is in feed mode
         RunMode { ExternalAccessible := 'False'; ExternalVisible := 'False'; ExternalWritable := 'False'} : Bool;   // Extendable is in run mode
      END_STRUCT;
   END_STRUCT;

END_TYPE

TYPE "UDT_PneumaticBrakeConfiguration"
VERSION : 0.1
   STRUCT
      BrakePuls : UDInt;   // Time [ms] brake is up in brake function
      BrakePause : UDInt;   // Time [ms] brake is down in brake function
      BrakeCycles : Int;   // Number of brake cycles
      BrakeInterval : UDInt;   // Time [ms] between brake cycles
      PECBrakeOnDelay : UDInt;   // On delay time PEC brake signal
      PECBrakeOffDelay : UDInt;   // Off delay time PEC brake signal
      PECStopOnDelay : UDInt;   // On delay time PEC stop signal
      PECStopOffDelay : UDInt;   // Off delay time PEC stop signal
      StopFunctionOnDelay : UDInt;   // On delay time stop function
      StopFunctionOffDelay : UDInt;   // Off delay time stop function
      FailSafe { ExternalAccessible := 'False'; ExternalVisible := 'False'; ExternalWritable := 'False'} : Bool;   // Activate output to release
      Slave { ExternalAccessible := 'False'; ExternalVisible := 'False'; ExternalWritable := 'False'} : Bool;   // Stopper is slave
   END_STRUCT;

END_TYPE

TYPE "UDT_ZPAinterface"
VERSION : 0.1
   STRUCT
      CommonStatus { S7_SetPoint := 'False'} : "UDT_CommonStatus";
      ConveyorInterface { S7_SetPoint := 'False'} : "UDT_ConveyorInterface";
      Handshake { S7_SetPoint := 'False'} : "UDT_ConveyorHandshake";
   END_STRUCT;

END_TYPE

TYPE "UDT_PendantVT100Configuration"
VERSION : 0.1
//Configuration variables for PendantVT100
   STRUCT
      Line1Cursor : Array[0..7] of Byte := [16#001B, 16#005B, 16#0031, 16#003B, 16#0033, 16#0048, 16#006D, 16#0000];   // Configuration of telegram command to move cursor to line 1
      Line2Cursor : Array[0..7] of Byte := [16#001B, 16#005B, 16#0032, 16#003B, 16#0035, 16#0048, 16#006D, 16#0000];   // Configuration of telegram command to move cursor to line 2
      DisplayName : String[8];   // PLC name with a max of 8 characters
      HornRequest { ExternalAccessible := 'False'; ExternalVisible := 'False'; ExternalWritable := 'False'} : Bool;   // True = Request horn to sound before VFD run
      PNDeviceName : String;   // Device name of pendant receiver
   END_STRUCT;

END_TYPE

TYPE "UDT_LoaderConfiguration"
TITLE = UDT_LoaderConfiguration
VERSION : 0.1
//User-defined structure of loader parameters.
   STRUCT
      PEC_EoSTimeOnDelay : UDInt;   // Photo eye time on delay
      PEC_EoSTimeOffDelay : UDInt;   // Photo eye time off delay
      CascadeTimeOnDelay : UDInt;   // Cascade time on delay
      Speedsetpoint : Int;   // Speedsetpoint: 0=Low, 1=Nom, 2=High
      EnergySaveLength : Int;   // Distance conveyor travelled before energy save activate [cm]
      Energy { ExternalAccessible := 'False'; ExternalVisible := 'False'; ExternalWritable := 'False'} : Bool;   // Energy save mode enable
   END_STRUCT;

END_TYPE

TYPE "UDT_PendantVT100InBytes"
VERSION : 0.1
   STRUCT
      StartButton1 { ExternalAccessible := 'False'; ExternalVisible := 'False'; ExternalWritable := 'False'} : Bool;   // start button pressed half way
      StartButton2 { ExternalAccessible := 'False'; ExternalVisible := 'False'; ExternalWritable := 'False'} : Bool;   // start button pressed full way
      Stop_NO { ExternalAccessible := 'False'; ExternalVisible := 'False'; ExternalWritable := 'False'} : Bool;   // NO contact of stop button
      Spare1 { ExternalAccessible := 'False'; ExternalVisible := 'False'; ExternalWritable := 'False'} : Bool;   // spare
      Spare2 { ExternalAccessible := 'False'; ExternalVisible := 'False'; ExternalWritable := 'False'} : Bool;   // spare
      Spare3 { ExternalAccessible := 'False'; ExternalVisible := 'False'; ExternalWritable := 'False'} : Bool;   // spare
      Spare4 { ExternalAccessible := 'False'; ExternalVisible := 'False'; ExternalWritable := 'False'} : Bool;   // spare
      Stop_NC { ExternalAccessible := 'False'; ExternalVisible := 'False'; ExternalWritable := 'False'} : Bool;   // NC contact of stop button
      LeftButton1 { ExternalAccessible := 'False'; ExternalVisible := 'False'; ExternalWritable := 'False'} : Bool;   // left button pressed half way
      PB_Speed2 { ExternalAccessible := 'False'; ExternalVisible := 'False'; ExternalWritable := 'False'} : Bool;   // Push button for low speed
      RightButton1 { ExternalAccessible := 'False'; ExternalVisible := 'False'; ExternalWritable := 'False'} : Bool;   // right button pressed half way
      PB_Speed1 { ExternalAccessible := 'False'; ExternalVisible := 'False'; ExternalWritable := 'False'} : Bool;   // Push button for manual speed
      DownButton1 { ExternalAccessible := 'False'; ExternalVisible := 'False'; ExternalWritable := 'False'} : Bool;   // down button pressed half way
      DownButton2 { ExternalAccessible := 'False'; ExternalVisible := 'False'; ExternalWritable := 'False'} : Bool;   // down button pressed full way
      UpButton1 { ExternalAccessible := 'False'; ExternalVisible := 'False'; ExternalWritable := 'False'} : Bool;   // up button pressed half way
      PB_Divert { ExternalAccessible := 'False'; ExternalVisible := 'False'; ExternalWritable := 'False'} : Bool;   // Push button to activate divert
      ResetButton1 { ExternalAccessible := 'False'; ExternalVisible := 'False'; ExternalWritable := 'False'} : Bool;   // reset button pressed half way
      ResetButton2 { ExternalAccessible := 'False'; ExternalVisible := 'False'; ExternalWritable := 'False'} : Bool;   // reset button pressed full way
      MOT_Button1 { ExternalAccessible := 'False'; ExternalVisible := 'False'; ExternalWritable := 'False'} : Bool;   // motor button pressed half way
      MOT_Button2 { ExternalAccessible := 'False'; ExternalVisible := 'False'; ExternalWritable := 'False'} : Bool;   // motor button pressed full way
      Spare5 { ExternalAccessible := 'False'; ExternalVisible := 'False'; ExternalWritable := 'False'} : Bool;   // spare
      Spare6 { ExternalAccessible := 'False'; ExternalVisible := 'False'; ExternalWritable := 'False'} : Bool;   // spare
      Spare7 { ExternalAccessible := 'False'; ExternalVisible := 'False'; ExternalWritable := 'False'} : Bool;   // spare
      Spare8 { ExternalAccessible := 'False'; ExternalVisible := 'False'; ExternalWritable := 'False'} : Bool;   // spare
   END_STRUCT;

END_TYPE

TYPE "UDT_PendantVT100LCDOutBytes"
VERSION : 0.1
   STRUCT
      "Byte" : Array[0..7] of Byte;   // Output byte for VT100 LCD
   END_STRUCT;

END_TYPE

TYPE "UDT_PendantVT100Status"
VERSION : 0.1
//Configuation variables for VT100 Radio Pendant
   STRUCT
      Status : Int;   // Status number
      Specific : Struct   // Specific structure
         PNSlaveNotOnline { ExternalAccessible := 'False'; ExternalVisible := 'False'; ExternalWritable := 'False'} : Bool;   // Profinet slave is not online
         PNSlaveError { ExternalAccessible := 'False'; ExternalVisible := 'False'; ExternalWritable := 'False'} : Bool;   // Profinet slave is in error
         CommunicationError { ExternalAccessible := 'False'; ExternalVisible := 'False'; ExternalWritable := 'False'} : Bool;   // Tx-Rx Communication error
         ServiceModeEngaged { ExternalAccessible := 'False'; ExternalVisible := 'False'; ExternalWritable := 'False'} : Bool;   // Service mode is activated
      END_STRUCT;
   END_STRUCT;

END_TYPE

TYPE "UDT_ValveCommand"
TITLE = UDT_ConveyorCommand
VERSION : 0.1
//User-defined structure of conveyor commands.
   STRUCT
      ManualMode { ExternalAccessible := 'False'; ExternalVisible := 'False'; ExternalWritable := 'False'} : Bool;   // Manual mode command from HMI
      AutoMode { ExternalAccessible := 'False'; ExternalVisible := 'False'; ExternalWritable := 'False'} : Bool;   // Automatic mode command from HMI
      ManualOpen { ExternalAccessible := 'False'; ExternalVisible := 'False'; ExternalWritable := 'False'} : Bool;   // Manual command valve Open / Extend
      ManualClose { ExternalAccessible := 'False'; ExternalVisible := 'False'; ExternalWritable := 'False'} : Bool;   // Manual command valve Close / Retract
   END_STRUCT;

END_TYPE

TYPE "UDT_ValveInterface"
TITLE = UDT_ValveInterface
VERSION : 0.1
//UDT valve interface between modules
   STRUCT
      Open { ExternalAccessible := 'False'; ExternalVisible := 'False'; ExternalWritable := 'False'} : Bool;   // Interface command valve Open / Extend
      Close { ExternalAccessible := 'False'; ExternalVisible := 'False'; ExternalWritable := 'False'} : Bool;   // Interface command valve Close / Retract
      IsOpened { ExternalAccessible := 'False'; ExternalVisible := 'False'; ExternalWritable := 'False'} : Bool;   // Valve feedback opened / extended
      IsClosed { ExternalAccessible := 'False'; ExternalVisible := 'False'; ExternalWritable := 'False'} : Bool;   // Valve feedback closed / retracted
      Error { ExternalAccessible := 'False'; ExternalVisible := 'False'; ExternalWritable := 'False'} : Bool;   // Valve error
   END_STRUCT;

END_TYPE

TYPE "UDT_FlowConfiguration"
VERSION : 0.1
   STRUCT
      FactorMerges : Array[1..6] of Real := [6(1.0)];
      MiniumGap : Int := 500;   // Minimum Gap setting [mm]
      MaxGap : Int := 2000;   // Maximum Gap setting [mm]
      PeriodSorterCapacity : UDInt := 30;   // Time  to check average empty carriers [s]
      PeriodMergeCapacity : UDInt := 30;   // Timer to check average merge flow [s]
      MaxCapacityMerge : Int;   // Max capacity Merge
   END_STRUCT;

END_TYPE

FUNCTION_BLOCK "FB_MergeGenerator"
TITLE = FB_BasicEquipment
{ S7_Optimized_Access := 'TRUE' }
AUTHOR : MHSE
FAMILY : Equipment
VERSION : 3.0
// ATTRIBUTES
// AUTO_NUMBER = True
// BLOCK_NUMBER = 17
// END_ATTRIBUTES
//Function block to control basic equipment.
   VAR_INPUT
      iUDT_MergeGenConfig { ExternalAccessible := 'False'; ExternalVisible := 'False'; ExternalWritable := 'False'} : "UDT_MergeGeneratorConfig";   // Merge configuration structure
      ii_ConveyorDisplacement { ExternalAccessible := 'False'; ExternalVisible := 'False'; ExternalWritable := 'False'} : Int;   // Displacement of merge conveyor
   END_VAR

   VAR_IN_OUT
      iqa_TrackingData : Array[*] of Int;   //  UDT Equipment Control
      iqUDT_Merge : "UDT_Merge";   // UDT Mergedata
      iqUDT_Induct : Array[*] of "UDT_Induct";   // UDT induct
   END_VAR

   VAR
      sR_TRIG_Full {InstructionName := 'R_TRIG'; LibVersion := '1.0'; ExternalAccessible := 'False'; ExternalVisible := 'False'; ExternalWritable := 'False'; S7_SetPoint := 'False'} : R_TRIG;
      sdi_DeactivateDistance { ExternalAccessible := 'False'; ExternalVisible := 'False'; ExternalWritable := 'False'} : DInt;   //  Distance to go before generator deactivates
      si_LoopCounterZero { ExternalAccessible := 'False'; ExternalVisible := 'False'; ExternalWritable := 'False'} : Int;   //  Loop Counter to delete empty positons
      si_GenerationGapCounter { ExternalAccessible := 'False'; ExternalVisible := 'False'; ExternalWritable := 'False'} : Int;   //  Generate the gap unit in the trackind DB
      si_LastInductNumberUsed { ExternalAccessible := 'False'; ExternalVisible := 'False'; ExternalWritable := 'False'} : Int;   //  Last Induct number used
      si_ReturnValue { ExternalAccessible := 'False'; ExternalVisible := 'False'; ExternalWritable := 'False'} : Int;   //  Info Code of Move Block Siemens
      si_GenerationPoint { ExternalAccessible := 'False'; ExternalVisible := 'False'; ExternalWritable := 'False'} : Int;   //  Position in tracking at which the window will be generated
      si_NumerOfInduct { ExternalAccessible := 'False'; ExternalVisible := 'False'; ExternalWritable := 'False'} : Int;   //  Number of inducts connected to the merge
      si_PositionsPerInduct { ExternalAccessible := 'False'; ExternalVisible := 'False'; ExternalWritable := 'False'} : Int;   //  Number of positions each induct has
      si_LoopCounter { ExternalAccessible := 'False'; ExternalVisible := 'False'; ExternalWritable := 'False'} : Int;   // Loopcounter number of inducts
      si_SecondLoopCounter { ExternalAccessible := 'False'; ExternalVisible := 'False'; ExternalWritable := 'False'} : Int;   // Loopcounter number of inducts
      si_LastInductNumber { ExternalAccessible := 'False'; ExternalVisible := 'False'; ExternalWritable := 'False'} : Int;   // Last induct number
      sx_LoopAgain { ExternalAccessible := 'False'; ExternalVisible := 'False'; ExternalWritable := 'False'} : Bool;   // Last used position was removed, loop again to find next
      sx_ShiftRequest { ExternalAccessible := 'False'; ExternalVisible := 'False'; ExternalWritable := 'False'} : Bool;   //  Request to Shift
   END_VAR


BEGIN
	(*
	----------------------------------------------------------------------------------------

	Version history:
	Date        | Version   | Author        | Remark
	----------------------------------------------------------------------------------------
	26/09/2019  | 1.0       | M.Roijen      | first release TIA 15.1
	12/11/2019  | 3.0       | P.Majka       | 3.0 MHS library release TIA 15.1
	07/01/2020  | 3.1       | F.Baten       | Added RequesetInFifo handshake
	13/01/2020  | 3.2       | F.Baten       | Removed i_UDT_ConveyorConfiguration as it was not used anymore
	23/01/2020  | 3.3       | F.Baten       | Renumber region 5-4 to 4-5
	                                        | Removed deletion off negative GIN
	                                        | Added 1cm to GenerationGapCounter as it has to set the desired gap, before it set the start position of the next parcel
	                                        | Removed i_UDT_ConveyorConfiguration and i_UDT_PECConfiguration as they were not used anymore
	30/03/2022  | 3.4       | H.Rutkowski   | Mode 2 handling
	22/07/2022  | 3.5       | M.Piela       | Check number of induct and numer of positions in induct every cycle
	21/02/2023  | 4.0       | F.Baten       | 4.0 Release TIA 17.5
	*)
	//
	//  This block generates gaps and windows for merge principles
	//
	REGION 1 - Mode Change Gap Mode / Window Mode

	    // CHeck number of induct and numer of positions in induct
	    #si_NumerOfInduct := "FC_GetNrOfArrayEl"(#iqUDT_Induct);
	    #si_PositionsPerInduct := "FC_GetNrOfArrayEl"(#iqUDT_Induct[1].Position);

	    #si_GenerationPoint := DINT_TO_INT(#iUDT_MergeGenConfig.GenerationPoint / 10);

	    // activate generation when request from induct is received
	    IF #iqUDT_Merge.ReactivateReq
	    THEN
	        #iqUDT_Merge.GenerationInactive := FALSE;
	        #iqUDT_Merge.ReactivateReq := FALSE;
	        #sdi_DeactivateDistance := #iUDT_MergeGenConfig.ChangeWindowModeDistance / 10;
	    END_IF;

	    //Deactivate generation mode when no generation request or distance traveled to disable mode
	    //********************************************
	    // #iq_UDT_Merge.GenerationInactive := (#sdi_DeactivateDistance <= 0)
	    // AND NOT #iq_UDT_Merge.ReactivateReq;

	    IF #iqUDT_Merge.GenerationInactive
	    THEN
	        #si_GenerationGapCounter := #iUDT_MergeGenConfig.GapHeadToHead;
	    END_IF;

	END_REGION

	REGION 2 - Update/shift FIFO
	    //Get size of FIFO array (without the zero)
	    #iqUDT_Merge.MaxNumberofEntries := ("FC_GetNrOfArrayEl"(#iqUDT_Merge.FIFO) - 1);

	    // Handle shift request merge (FIFO entry is handled induct code is generated in tracking DB)
	    IF #sx_ShiftRequest
	    THEN
	        #si_ReturnValue := MOVE_BLK_VARIANT(SRC := #iqUDT_Merge.FIFO,
	                                            COUNT := INT_TO_UDINT(#iqUDT_Merge.MaxNumberofEntries),
	                                            SRC_INDEX := 1,
	                                            DEST_INDEX := 0,
	                                            DEST => #iqUDT_Merge.FIFO);
	        // reset the last entry and shift request
	        #iqUDT_Merge.FIFO[#iqUDT_Merge.MaxNumberofEntries].GapSize := 0;
	        #iqUDT_Merge.FIFO[#iqUDT_Merge.MaxNumberofEntries].InductNumber := 0;
	        #sx_ShiftRequest := False;

	        //Update last used position of FIFO.
	        #iqUDT_Merge.LastUsed -= 1;
	        IF #iqUDT_Merge.LastUsed < 0           // value can not be smaller than '0'
	        THEN
	            #iqUDT_Merge.LastUsed := 0;
	        END_IF;
	    END_IF;
	END_REGION

	REGION 3 - FIFO checks

	    REGION 3.1 - Remove '0' entry
	        IF NOT (#iUDT_MergeGenConfig.ModeSelection = 2)
	        THEN
	            // There was an entry removed by one of the inducts (remove is true)
	            // now the 'RemoveEntry' is searched for and if found deleted from the FIFO by shifting up
	            IF #iqUDT_Merge.Remove OR #sx_LoopAgain
	            THEN
	                // Loop again bit will be false until a RemoveEntry is found
	                #sx_LoopAgain := FALSE;

	                // check all entries for RemoveEntry = true
	                FOR #si_LoopCounterZero := 1 TO #iqUDT_Merge.MaxNumberofEntries BY 1 DO
	                    IF #iqUDT_Merge.FIFO[#si_LoopCounterZero].RemoveEntry
	                    THEN
	                        #si_ReturnValue := MOVE_BLK_VARIANT(SRC := #iqUDT_Merge.FIFO,
	                                                            COUNT := INT_TO_UDINT(#iqUDT_Merge.MaxNumberofEntries - #si_LoopCounterZero),
	                                                            SRC_INDEX := #si_LoopCounterZero + 1,
	                                                            DEST_INDEX := #si_LoopCounterZero,
	                                                            DEST => #iqUDT_Merge.FIFO);
	                        // reset the last entry if shift is executed
	                        #iqUDT_Merge.FIFO[#iqUDT_Merge.MaxNumberofEntries].GapSize := 0;
	                        #iqUDT_Merge.FIFO[#iqUDT_Merge.MaxNumberofEntries].InductNumber := 0;
	                        #iqUDT_Merge.FIFO[#iqUDT_Merge.MaxNumberofEntries].RemoveEntry := FALSE;

	                        //Update Last Used position of FIFO.
	                        #iqUDT_Merge.LastUsed -= 1;
	                        #iqUDT_Merge.Remove := FALSE;
	                        #sx_LoopAgain := TRUE;
	                    END_IF;
	                    IF #si_LoopCounterZero = #iqUDT_Merge.MaxNumberofEntries
	                        AND #iqUDT_Merge.Remove
	                    THEN
	                        #iqUDT_Merge.Remove := FALSE;
	                    END_IF;
	                END_FOR;
	                // Checking if last used value does not go below 0, if so, write back to 0
	                IF #iqUDT_Merge.LastUsed < 0
	                THEN
	                    #iqUDT_Merge.LastUsed := 0;
	                END_IF;
	            END_IF;
	        END_IF;
	    END_REGION

	    REGION 3.2 - Check if last used bit is accurate and correct if it is not.
	        // Last used can't be an empty entry unless it is equal to '0'
	        IF #iqUDT_Merge.FIFO[#iqUDT_Merge.LastUsed].InductNumber = 0
	            AND #iqUDT_Merge.LastUsed <> 0
	        THEN
	            #iqUDT_Merge.LastUsed -= 1;
	        END_IF;

	        // When the next entry is filled then the number has to be increased
	        IF #iqUDT_Merge.LastUsed < #iqUDT_Merge.MaxNumberofEntries
	        THEN
	            IF #iqUDT_Merge.FIFO[#iqUDT_Merge.LastUsed].InductNumber <> 0
	                AND #iqUDT_Merge.FIFO[#iqUDT_Merge.LastUsed + 1].InductNumber <> 0
	            THEN
	                #iqUDT_Merge.LastUsed += 1;
	            END_IF;
	        END_IF;
	    END_REGION
	END_REGION

	REGION 4 - Update on displacement
	    // decrease the gap counter as long the gap counter is bigger than '0'
	    IF #si_GenerationGapCounter > 0
	    THEN
	        #si_GenerationGapCounter -= #ii_ConveyorDisplacement;

	        // check if value does not go negative
	        IF #si_GenerationGapCounter < 0
	        THEN
	            #si_GenerationGapCounter := 0;
	        END_IF;
	    END_IF;

	    // decrease the deactivation distance counter as long as it is bigger than '0'
	    IF #sdi_DeactivateDistance > 0
	    THEN
	        #sdi_DeactivateDistance -= #ii_ConveyorDisplacement;

	        // check if value does not go negative
	        IF #sdi_DeactivateDistance < 0
	        THEN
	            #sdi_DeactivateDistance := 0;
	        END_IF;
	    END_IF;

	    IF (#iUDT_MergeGenConfig.ModeSelection = 2)
	        AND NOT #iqUDT_Merge.GenerationInactive
	        AND #ii_ConveyorDisplacement > 0
	    THEN
	        FOR #si_LoopCounter := 1 TO #si_NumerOfInduct DO
	            #iqUDT_Induct[#si_LoopCounter].DistanceLastReserved -= #ii_ConveyorDisplacement;
	            IF #iqUDT_Induct[#si_LoopCounter].DistanceLastReserved < 0
	            THEN
	                #iqUDT_Induct[#si_LoopCounter].DistanceLastReserved := 0;
	            END_IF;
	        END_FOR;
	    END_IF;
	END_REGION

	REGION 5 - Put Value in Tracking array
	    // check if required gap is reached and if the generation is active
	    REGION Mode 0 and 1
	        IF (#si_GenerationGapCounter = 0)
	            AND NOT #iqUDT_Merge.GenerationInactive
	            AND NOT (#iUDT_MergeGenConfig.ModeSelection = 2)
	        THEN
	            // check if FIFO does contain requests to generate induct codes
	            IF #iqUDT_Merge.FIFO[1].InductNumber = 0 AND #iUDT_MergeGenConfig.ModeSelection = 0
	            THEN
	                // If no request generate value -100 in tracking DB with the correpondent fixed window, and set counter to create gap.
	                #iqa_TrackingData[#si_GenerationPoint] := -100;
	                #si_GenerationGapCounter := #iUDT_MergeGenConfig.GapHeadToHead;
	            END_IF;

	            IF #iqUDT_Merge.FIFO[1].InductNumber > 0
	                AND NOT #sx_ShiftRequest
	            THEN
	                // If there is assigned a induct number add 100 and negate the value.
	                // Move the position value into the tracking request variable
	                // Inform that the request was handled.
	                #iqa_TrackingData[#si_GenerationPoint] := - (#iqUDT_Merge.FIFO[1].InductNumber + 100);
	                #iqUDT_Merge.TrackingPointerForInduct[#iqUDT_Merge.FIFO[1].InductNumber] := #si_GenerationPoint;
	                #iqUDT_Merge.RequestInFIFO[#iqUDT_Merge.FIFO[1].InductNumber] := FALSE;

	                // Compares the last entry to be different to 0 and to the actual entry , if they are set the distance.
	                IF (#si_LastInductNumberUsed <> #iqa_TrackingData[#si_GenerationPoint])
	                THEN
	                    #sdi_DeactivateDistance := #iUDT_MergeGenConfig.ChangeWindowModeDistance / 10;
	                END_IF;

	                // write last induct number used to static for next compare
	                #si_LastInductNumberUsed := #iqa_TrackingData[#si_GenerationPoint];

	                // initiate gap counter and set shift request
	                #si_GenerationGapCounter := (#iqUDT_Merge.FIFO[1].GapSize + 1);
	                #sx_ShiftRequest := TRUE;

	            END_IF;
	        END_IF;
	    END_REGION

	    REGION Mode = 2
	        // Statement section REGION
	        IF (#iUDT_MergeGenConfig.ModeSelection = 2)
	            AND NOT #iqUDT_Merge.GenerationInactive
	            AND (#si_GenerationGapCounter = 0)
	        THEN

	            //generate window from last induct to 1st induct
	            FOR #si_SecondLoopCounter := 1 TO #si_NumerOfInduct DO

	                IF #si_LastInductNumber <= 1
	                THEN
	                    #si_LastInductNumber := #si_NumerOfInduct + 1;

	                END_IF;

	                #si_LastInductNumber := #si_LastInductNumber - 1;


	                // Check induct buffer conveyor for which window need to be reserved

	                IF #iqUDT_Induct[#si_LastInductNumber].DistanceLastReserved <= 0 AND
	                    NOT #iqUDT_Induct[#si_LastInductNumber].DisableWindowReservation
	                THEN
	                    FOR #si_LoopCounter := 1 TO #si_PositionsPerInduct DO
	                        IF #iqUDT_Induct[#si_LastInductNumber].Position[#si_LoopCounter].GapRequired > 0
	                            AND #iqUDT_Induct[#si_LastInductNumber].Position[#si_LoopCounter].GINNumber > 0
	                            AND NOT #iqUDT_Induct[#si_LastInductNumber].Position[#si_LoopCounter].WindowReserved
	                        THEN
	                            #iqa_TrackingData[#si_GenerationPoint] := - (#si_LastInductNumber + 100);
	                            #iqa_TrackingData[#si_GenerationPoint + 1] := #iqUDT_Induct[#si_LastInductNumber].Position[#si_LoopCounter].GapRequired;
	                            //Test code, write GIN number into tracking array
	                            #iqa_TrackingData[#si_GenerationPoint + 2] := #iqUDT_Induct[#si_LastInductNumber].Position[#si_LoopCounter].GINNumber;

	                            #iqUDT_Induct[#si_LastInductNumber].Position[#si_LoopCounter].WindowPosition := #si_GenerationPoint;
	                            #iqUDT_Induct[#si_LastInductNumber].Position[#si_LoopCounter].WindowReserved := TRUE;
	                            #si_GenerationGapCounter := #iqUDT_Induct[#si_LastInductNumber].Position[#si_LoopCounter].GapRequired;
	                            #iqUDT_Induct[#si_LastInductNumber].DistanceLastReserved := #iUDT_MergeGenConfig.DelayDistance;

	                            // Compares the last entry to be different to 0 and to the actual entry , if they are set the distance.
	                            IF (#si_LastInductNumberUsed <> #si_LastInductNumber)
	                            THEN
	                                #sdi_DeactivateDistance := #iUDT_MergeGenConfig.ChangeWindowModeDistance / 10;
	                            END_IF;

	                            // write last induct number used to static for next compare
	                            #si_LastInductNumberUsed := #si_LastInductNumber;

	                            EXIT;
	                        END_IF;
	                        IF #iqUDT_Induct[#si_LastInductNumber].Position[#si_LoopCounter].GINNumber = 0
	                        THEN
	                            EXIT;
	                        END_IF;
	                    END_FOR;
	                END_IF;
	                IF #si_GenerationGapCounter > 0
	                THEN
	                    EXIT;
	                END_IF;
	            END_FOR;
	        END_IF;

	    END_REGION

	END_REGION
END_FUNCTION_BLOCK

FUNCTION "FC_NordToSiemensVFDSimulationOutput" : Void
{ S7_Optimized_Access := 'TRUE' }
VERSION : 0.1
// ATTRIBUTES
// AUTO_NUMBER = True
// BLOCK_NUMBER = 24
// END_ATTRIBUTES
   VAR_INPUT
      qUDT_VfdOutputsNord : "UDT_VfdNordPO";
   END_VAR

   VAR_OUTPUT
      qUDT_VfdOutputsSiemens : "UDT_VfdSiemensPO";
   END_VAR

   VAR_TEMP
      tx_dummy : Bool;
      ti_dummy : Int;
   END_VAR


BEGIN
	(*
	----------------------------------------------------------------------------------------

	Version history:
	Date        | Version   | Author        | Remark
	----------------------------------------------------------------------------------------
	24/11/2021  | 0.1       | M.Roijen      | Initial version TIA 15.1
	21/02/2023  | 4.0       | F.Baten       | 4.0 Release TIA 17.5
	*)

	REGION 1 - Send VFD Output to Siemens Drive

	    #qUDT_VfdOutputsSiemens.STW_1.ControlViaPLC := TRUE;
	    #qUDT_VfdOutputsSiemens.STW_1.DirectionReversal := FALSE;
	    #qUDT_VfdOutputsSiemens.STW_1.ONOFF1 := #qUDT_VfdOutputsNord.STW.ReadyForOperation;
	    #qUDT_VfdOutputsSiemens.STW_1.OFF2 := TRUE;
	    #qUDT_VfdOutputsSiemens.STW_1.OFF3 := #qUDT_VfdOutputsNord.STW.EmergencyStop;
	    #qUDT_VfdOutputsSiemens.STW_1.EnableOperation := #qUDT_VfdOutputsNord.STW.ReadyForOperation;
	    #qUDT_VfdOutputsSiemens.STW_1.EnableSetpoint := TRUE;
	    #qUDT_VfdOutputsSiemens.SpeedSetpoint := #qUDT_VfdOutputsNord.FrequencySetPoint;
	    #qUDT_VfdOutputsSiemens.SetpointAcceleration := #qUDT_VfdOutputsNord.RampTimeSetPoint * 2;  //#cr_MaximumOutput is 16384 in siemens and 32676 in Nord drive
	    #qUDT_VfdOutputsSiemens.SetpointDeceleration := #qUDT_VfdOutputsNord.RampTimeSetPoint * 2; //#cr_MaximumOutput is 16384 in siemens and 32676 in Nord drive

	END_REGION


END_FUNCTION

FUNCTION "FC_InterPLCHandshake" : Void
TITLE = Interconnection PLC Handshake
{ S7_Optimized_Access := 'TRUE' }
AUTHOR : MHSE
VERSION : 3.0
// ATTRIBUTES
// AUTO_NUMBER = True
// BLOCK_NUMBER = 22
// END_ATTRIBUTES
   VAR_INPUT
      iUDT_HandshakeInput : "UDT_PNCoupler_Interface";   // Input bytes from PN Coupler to the PLC
      ix_ConfigUpstream : Bool;   // True = Conveyor is the upstream conveyor; False = Conveyor is the downstream conveyor.
   END_VAR

   VAR_OUTPUT
      qUDT_HandshakeOutput : "UDT_PNCoupler_Interface";   // Output bytes from PLC to the PN Coupler
   END_VAR

   VAR_IN_OUT
      iqUDT_HandshakeDB : "UDT_ConveyorHandshake";   // Handshake Database
   END_VAR


BEGIN
	(*
	----------------------------------------------------------------------------------------

	Version history:
	Date        | Version   | Author        | Remark
	----------------------------------------------------------------------------------------
	30/09/2019  | 2.1       | C. Leite      | first release MHS TIA 15.1
	09/10/2019  | 2.2       | C. Leite      | Bug correction
	04/11/2019  | 2.3       | C. Leite      | New PN Coupler handshake
	12/11/2019  | 3.0       | P.Majka       | 3.0 MHS library release TIA 15.1
	21/02/2023  | 4.0       | F.Baten       | 4.0 Release TIA 17.5
	*)

	REGION 1 - Downstream Configuration Inputs

	    IF NOT #ix_ConfigUpstream
	    THEN

	        #iqUDT_HandshakeDB.RTS := #iUDT_HandshakeInput.RTS;
	        #iqUDT_HandshakeDB.TIP := #iUDT_HandshakeInput.TIP;
	        #iqUDT_HandshakeDB.ResetEnergySave := #iUDT_HandshakeInput.ResetEnergySave;

	    END_IF;

	END_REGION

	REGION 2 - Downstream Configuration Outputs

	    IF NOT #ix_ConfigUpstream
	    THEN

	        #qUDT_HandshakeOutput.DownstreamDisplacement := #iqUDT_HandshakeDB.DownstreamDisplacement;
	        #qUDT_HandshakeOutput.RTR := #iqUDT_HandshakeDB.RTR;
	        #qUDT_HandshakeOutput.CascadeStartUp := #iqUDT_HandshakeDB.CascadeStartUp;

	    END_IF;

	END_REGION

	REGION 3 - Upstream Configuration Inputs

	    IF #ix_ConfigUpstream
	    THEN

	        #iqUDT_HandshakeDB.DownstreamDisplacement := #iUDT_HandshakeInput.DownstreamDisplacement;
	        #iqUDT_HandshakeDB.RTR := #iUDT_HandshakeInput.RTR;
	        #iqUDT_HandshakeDB.CascadeStartUp := #iUDT_HandshakeInput.CascadeStartUp;

	    END_IF;

	END_REGION

	REGION 4 - Upstream Configuration Outputs

	    IF #ix_ConfigUpstream
	    THEN

	        #qUDT_HandshakeOutput.RTS := #iqUDT_HandshakeDB.RTS;
	        #qUDT_HandshakeOutput.TIP := #iqUDT_HandshakeDB.TIP;
	        #qUDT_HandshakeOutput.ResetEnergySave := #iqUDT_HandshakeDB.ResetEnergySave;

	    END_IF;

	END_REGION


END_FUNCTION

FUNCTION_BLOCK "FB_InductSpeedControl"
{ S7_Optimized_Access := 'TRUE' }
VERSION : 0.1
// ATTRIBUTES
// AUTO_NUMBER = True
// BLOCK_NUMBER = 16
// END_ATTRIBUTES
   VAR_INPUT
      ix_PEC { ExternalAccessible := 'False'; ExternalVisible := 'False'; ExternalWritable := 'False'} : Bool;   // Filtred signal of the PEC
      idiPEC_EoSDistance { ExternalAccessible := 'False'; ExternalVisible := 'False'; ExternalWritable := 'False'} : DInt;   // Distance between photo eye and the end of conveyor [mm] in forward direction
      ii_TrackingEndPosition { ExternalAccessible := 'False'; ExternalVisible := 'False'; ExternalWritable := 'False'} : Int;   // Position of the tracking in the end of the conveyor
      ii_SpeedSetpointHigh { ExternalAccessible := 'False'; ExternalVisible := 'False'; ExternalWritable := 'False'} : Int;   // Speed setpoint High [mm/s]
      ii_SpeedSetpointLow { ExternalAccessible := 'False'; ExternalVisible := 'False'; ExternalWritable := 'False'} : Int;   // Speed setpoint Low [mm/s]
   END_VAR

   VAR_OUTPUT
      qi_Speed { ExternalAccessible := 'False'; ExternalVisible := 'False'; ExternalWritable := 'False'} : Int;
   END_VAR

   VAR_IN_OUT
      iqi_Displacement { ExternalAccessible := 'False'; ExternalVisible := 'False'; ExternalWritable := 'False'} : Int;   // Displacement per PLC scan [cm]
   END_VAR

   VAR
      sR_TRIG_PEC {InstructionName := 'R_TRIG'; LibVersion := '1.0'; ExternalAccessible := 'False'; ExternalVisible := 'False'; ExternalWritable := 'False'; S7_SetPoint := 'False'} : R_TRIG;
      sdi_ParcelTailAtEnd { ExternalAccessible := 'False'; ExternalVisible := 'False'; ExternalWritable := 'False'} : DInt;   // Count tail to next conveyor distance
      sx_PEC { ExternalAccessible := 'False'; ExternalVisible := 'False'; ExternalWritable := 'False'} : Bool;   // Auxiliary variable when the PEC detect the parcel
      sx_ParcelTailAtEnd { ExternalAccessible := 'False'; ExternalVisible := 'False'; ExternalWritable := 'False'} : Bool;   // Tail at the end of the conveyor
   END_VAR


BEGIN
	(*
	----------------------------------------------------------------------------------------

	Version history:
	Date        | Version   | Author        | Remark
	----------------------------------------------------------------------------------------
	24/02/2022  | 3.0       | M.Piela       | First release TIA 16.1
	17/02/2023  | 3.1       | F.Baten       | Added regions
	21/02/2023  | 4.0       | F.Baten       | 4.0 Release TIA 17.5
	*)

	REGION 1 - Initial
	    // Low speed at startup
	    IF "DB_Memory".FirstScan
	    THEN
	        #qi_Speed := #ii_SpeedSetpointLow;
	    END_IF;

	END_REGION

	REGION 2 - Triggers
	    // Rising trigger PEC
	    #sR_TRIG_PEC(CLK := #ix_PEC);

	END_REGION

	REGION 3 - Distance

	    //Check if the parcel travels at the end of the conveyor
	    IF #sR_TRIG_PEC.Q AND (#sdi_ParcelTailAtEnd <= 0)
	    THEN
	        #sdi_ParcelTailAtEnd := (#idiPEC_EoSDistance / 10);
	    END_IF;

	    IF #sdi_ParcelTailAtEnd > 0
	    THEN
	        #sdi_ParcelTailAtEnd -= #iqi_Displacement;
	        #sx_ParcelTailAtEnd := FALSE;
	    ELSE
	        #sx_ParcelTailAtEnd := TRUE;
	    END_IF;
	END_REGION


	REGION 4 - Control speed

	    //When the parcel reach the end of the conveyor are in the last tracking number is no data then set the low speed.
	    IF (#sx_ParcelTailAtEnd AND (#ii_TrackingEndPosition = 0))
	    THEN
	        #qi_Speed := #ii_SpeedSetpointLow;
	    END_IF;

	    // Set the High after detecting parcel on the photo cell
	    IF #sR_TRIG_PEC.Q
	    THEN
	        #qi_Speed := #ii_SpeedSetpointHigh;

	    END_IF;
	END_REGION








END_FUNCTION_BLOCK

FUNCTION "FC_SeparateMsg" : Void
TITLE = FC_SeparateMsg
{ S7_Optimized_Access := 'TRUE' }
AUTHOR : MHSE
FAMILY : GeneralSystemFunctions
VERSION : 3.0
// ATTRIBUTES
// AUTO_NUMBER = True
// BLOCK_NUMBER = 25
// END_ATTRIBUTES
//Function to separate the delimited message.
   VAR_INPUT
      iUDT_Message : "UDT_Message";   // Character string to be separated
      ii_Position : Int;   // Start position
      ic_Delimiter : Char;   // Delimiter
      ic_EndSign : Char;   // End of the message sign
   END_VAR

   VAR_OUTPUT
      qs_Msg : String;   // Separated part of the message
      qui_Length : UInt;   // Length of the separated message
      qx_EndMsg : Bool;   // End message sign found
      qx_NoSeparationSign : Bool;   // Separation sign not detected
   END_VAR

   VAR_TEMP
      ti_i : Int;   // Loop counter
      tui_NrOfConvChar : UInt;   // Number of converted message characters
      ti_SizeOfMsg : Int;   // Message array size
   END_VAR


BEGIN
	(*
	----------------------------------------------------------------------------------------

	Version history:
	Date        | Version   | Author        | Remark
	----------------------------------------------------------------------------------------
	24/05/2019  | 0.1       | K.Pokorski    | first release MHS TIA 15.1
	14/06/2019  | 0.2       | K.Pokorski    | "ii_Position" input, "qx_NoSeparationSign" output added, additional logic programmed
	17/06/2019  | 0.3       | L.Klar        | "iqi_Position" deleted
	24/07/2019  | 2.0       | L.Klar        | 2.0 MHS library release TIA 15.1
	26/07/2019  | 2.1       | M.Kurpiers    | Comments adjusted
	12/11/2019  | 3.0       | P.Majka       | 3.0 MHS library release TIA 15.1
	21/02/2023  | 4.0       | F.Baten       | 4.0 Release TIA 17.5
	*)

	REGION 1 – Maximum number of the message characters

	    #ti_SizeOfMsg := "FC_GetNrOfArrayEl"(iv_Array := #iUDT_Message.Character);

	END_REGION

	REGION 2 – Message separation

	    IF (#ii_Position <= #ti_SizeOfMsg - 1)                                        // Position is lower than size of a message array
	    THEN

	        // Delimiter and end sign search loop
	        FOR #ti_i := #ii_Position TO #ti_SizeOfMsg - 1 DO


	            IF (#iUDT_Message.Character[#ti_i] = #ic_Delimiter                    // Check if delimiter and the end of the message was found
	                OR #iUDT_Message.Character[#ti_i] = #ic_EndSign)

	            THEN

	                // Message length minus start position from INT to UInt conversion
	                #tui_NrOfConvChar := INT_TO_UINT(IN := (#ti_i - #ii_Position));

	                IF #tui_NrOfConvChar <> 0
	                THEN
	                    // Character array into the message character string conversion
	                    Chars_TO_Strg(Chars := #iUDT_Message.Character,
	                                  pChars := #ii_Position,
	                                  Cnt := #tui_NrOfConvChar,
	                                  Strg => #qs_Msg);

	                ELSE
	                    #qs_Msg := '';
	                END_IF;

	                // Length of the separated message part
	                #qui_Length := #tui_NrOfConvChar;

	                // Separation sign not detected
	                #qx_NoSeparationSign := FALSE;


	                IF (#iUDT_Message.Character[#ti_i] = #ic_EndSign)                   // End of the message sign detected
	                THEN

	                    #qx_EndMsg := TRUE;

	                ELSE

	                    #qx_EndMsg := FALSE;

	                END_IF;
	                // Exit the loop if end sign was found
	                EXIT;


	            ELSIF (#ti_i = #ti_SizeOfMsg - 1)                                         // Separate sign is not detected
	            THEN

	                // End of the message and no separation sign detected bits are set
	                #qs_Msg := '';
	                #qui_Length := 0;
	                #qx_EndMsg := TRUE;
	                #qx_NoSeparationSign := TRUE;

	            END_IF;

	        END_FOR;
	        // Clear variables if delimiter and end sign wasn't found
	    ELSE

	        #qs_Msg := '';
	        #qui_Length := 0;
	        #qx_EndMsg := TRUE;
	        #qx_NoSeparationSign := TRUE;

	    END_IF;

	END_REGION
END_FUNCTION

FUNCTION "FC_NordToSiemensVFDSimulationInput" : Void
{ S7_Optimized_Access := 'TRUE' }
VERSION : 0.1
// ATTRIBUTES
// AUTO_NUMBER = True
// BLOCK_NUMBER = 23
// END_ATTRIBUTES
   VAR_INPUT
      iUDT_VFDInputsSiemens : "UDT_VfdSiemensPI";
   END_VAR

   VAR_OUTPUT
      iUDT_VFDInputsNord : "UDT_VfdNordPI";
   END_VAR

   VAR_TEMP
      tx_dummy : Bool;
      ti_dummy : Int;
   END_VAR


BEGIN
	(*
	----------------------------------------------------------------------------------------

	Version history:
	Date        | Version   | Author        | Remark
	----------------------------------------------------------------------------------------
	24/11/2021  | 0.1       | M.Roijen      | Initial version TIA 15.1
	21/02/2023  | 4.0       | F.Baten       | 4.0 Release TIA 17.5
	*)

	REGION 1 - Get VFD input of Siemens drive

	    #iUDT_VFDInputsNord.ZSW.BusControlActive := TRUE;
	    #iUDT_VFDInputsNord.ZSW.ReadyToStart := TRUE;
	    #iUDT_VFDInputsNord.ZSW.OperationEnabled := TRUE;
	    #iUDT_VFDInputsNord.ZSW.EmergencyStop := FALSE;
	    #iUDT_VFDInputsNord.ZSW.Fault := #iUDT_VFDInputsSiemens.ZSW_1.FaultActive;
	    #iUDT_VFDInputsNord.ZSW.WarningActive := #iUDT_VFDInputsSiemens.ZSW_1.AlarmActive;
	    #iUDT_VFDInputsNord.ActualSpeed := #iUDT_VFDInputsSiemens.ActualSpeed;

	END_REGION




END_FUNCTION

FUNCTION "FC_TimeDiff" : Void
TITLE = FC_TimeDiff
{ S7_Optimized_Access := 'TRUE' }
AUTHOR : MHSE
FAMILY : GeneralSystemFunctions
VERSION : 3.0
// ATTRIBUTES
// AUTO_NUMBER = True
// BLOCK_NUMBER = 28
// END_ATTRIBUTES
//Function to calculate time difference.
   VAR_INPUT
      is_EarlierTimeAsString : String;   // Earlier time in string
      is_LaterTimeAsString : String;   // Later time in sting
   END_VAR

   VAR_OUTPUT
      qt_TimeDifference : LTime;   // Difference between times
   END_VAR

   VAR_TEMP
      tt_EarlierDate {InstructionName := 'DTL'; LibVersion := '1.0'} : DTL;   // Earlier date in DTL
      tt_LaterDate {InstructionName := 'DTL'; LibVersion := '1.0'} : DTL;   // Later date in DTL
      tt_LaterDateInc {InstructionName := 'DTL'; LibVersion := '1.0'} : DTL;   // Later date in DTL with one additional day
      tt_TimeDifference : LTime;   // Time differance
   END_VAR

   VAR CONSTANT
      ct_OneDay : Time := T#1D;   // One day
   END_VAR


BEGIN
	(*
	----------------------------------------------------------------------------------------

	Version history:
	Date        | Version   | Author        | Remark
	----------------------------------------------------------------------------------------
	24/05/2019  | 0.1       | K.Pokorski    | first release MHS TIA 15.1
	24/07/2019  | 2.0       | L.Klar        | 2.0 MHS library release TIA 15.1
	26/08/2019  | 2.1       | M.Kurpiers    | Comments adjusted
	06/09/2019  | 2.2       | M.Kurpiers    | Change in region 2. Correcting the names of inputs variables.
	21/10/2019  | 2.3       | P.Majka       | Logic changed in region 2 and 3. Simpler checking for the date changed
	12/11/2019  | 3.0       | P.Majka       | 3.0 MHS library release TIA 15.1
	21/02/2023  | 4.0       | F.Baten       | 4.0 Release TIA 17.5
	*)

	REGION 1 - Conversion string TO DTL

	    // Using MHS "FC_StringToTime" standard function convert time in string format to date in DTL format
	    "FC_StringToTime"(is_StringTime := #is_EarlierTimeAsString,
	                      qt_Date => #tt_EarlierDate);

	    "FC_StringToTime"(is_StringTime := #is_LaterTimeAsString,
	                      qt_Date => #tt_LaterDate);

	END_REGION

	REGION 2 - Difference between times

	    // Calculate difference between times
	    #tt_TimeDifference := #tt_LaterDate - #tt_EarlierDate;

	    // Checking the negativity in the time difference
	    IF (LTIME_TO_DINT(#tt_TimeDifference) < 0)
	    THEN

	        // Add one day to later date - later time is smaller than ealier time
	        #tt_LaterDateInc := T_ADD(IN1 := #tt_LaterDate, IN2 := #ct_OneDay);

	        // Calculate difference between times
	        #tt_TimeDifference := #tt_LaterDateInc - #tt_EarlierDate;

	    END_IF;

	END_REGION

	REGION 3 - Write outputs

	    // Saving time difference to the output
	    #qt_TimeDifference := #tt_TimeDifference;

	END_REGION
END_FUNCTION

FUNCTION_BLOCK "FB_ConveyorZPAlast"
{ S7_Optimized_Access := 'TRUE' }
VERSION : 0.1
   VAR_OUTPUT
      qUDT_CommonStatus { ExternalAccessible := 'False'; ExternalVisible := 'False'; ExternalWritable := 'False'} : "UDT_CommonStatus";   //           Common status structure
   END_VAR

   VAR_IN_OUT
      iqUDT_ConveyorInterface : "UDT_ConveyorInterface";   //           Handshake structure in forward direction
      iqUDT_ZPAinterface : "UDT_ZPAinterface";   //           Handshake structure in forward direction
      iqUDT_HandShake : "UDT_ConveyorHandshake";   //           Handshake structure in forward direction
   END_VAR

   VAR
      sUDT_HandShake { ExternalAccessible := 'False'; ExternalVisible := 'False'; ExternalWritable := 'False'; S7_SetPoint := 'False'} : "UDT_ConveyorHandshake";   //           Handshake structure in forward direction
   END_VAR


BEGIN
	(*
	----------------------------------------------------------------------------------------

	Version history:
	Date        | Version   | Author        | Remark
	----------------------------------------------------------------------------------------
	02/10/2024  | 1.0       | R.Willems     | First release TIA 18


	*)

	REGION 1 Common status
	    //Write
	    #qUDT_CommonStatus := #iqUDT_ZPAinterface.CommonStatus;
	END_REGION

	REGION 2 Conveyor interface
	    REGION 2.1 Displacement
	        //Write
	        //NOT USED, USES OWN DISPLACEMENT
	        //#iqUDT_ConveyorInterface.Displacement := #iqUDT_ZPAinterface.ConveyorInterface.Displacement;
	        #iqUDT_ConveyorInterface.ActualSpeed := #iqUDT_ZPAinterface.ConveyorInterface.ActualSpeed;
	    END_REGION
	    REGION 2.1 PEC
	        //Connect ZPA Interface to PEC
	        #iqUDT_ConveyorInterface.InternalErrorReset := #iqUDT_ZPAinterface.ConveyorInterface.InternalErrorReset;
	        #iqUDT_ConveyorInterface.ResetStatistics := #iqUDT_ZPAinterface.ConveyorInterface.ResetStatistics;
	        //Read
	        #iqUDT_ZPAinterface.ConveyorInterface.InternalErrorPEC := #iqUDT_ConveyorInterface.InternalErrorPEC;
	    END_REGION
	END_REGION

	REGION 3 Handshake
	    //Write
	    #iqUDT_HandShake.GIN := #sUDT_HandShake.GIN := #iqUDT_ZPAinterface.Handshake.GIN;
	    //Write/Read
	    IF #iqUDT_HandShake.RTS <> #sUDT_HandShake.RTS THEN
	        #iqUDT_ZPAinterface.Handshake.RTS := #sUDT_HandShake.RTS := #iqUDT_HandShake.RTS;
	    ELSE
	        #iqUDT_HandShake.RTS := #sUDT_HandShake.RTS := #iqUDT_ZPAinterface.Handshake.RTS;
	    END_IF;
	    IF #iqUDT_HandShake.RTR <> #sUDT_HandShake.RTR THEN
	        #iqUDT_ZPAinterface.Handshake.RTR := #sUDT_HandShake.RTR := #iqUDT_HandShake.RTR;
	    ELSE
	        #iqUDT_HandShake.RTR := #sUDT_HandShake.RTR := #iqUDT_ZPAinterface.Handshake.RTR;
	    END_IF;
	    IF #iqUDT_HandShake.TIP <> #sUDT_HandShake.TIP THEN
	        #iqUDT_ZPAinterface.Handshake.TIP := #sUDT_HandShake.TIP := #iqUDT_HandShake.TIP;
	    ELSE
	        #iqUDT_HandShake.TIP := #sUDT_HandShake.TIP := #iqUDT_ZPAinterface.Handshake.TIP;
	    END_IF;
	END_REGION


END_FUNCTION_BLOCK

FUNCTION_BLOCK "FB_Sensor"
TITLE = FB_PEC
{ S7_Optimized_Access := 'TRUE' }
AUTHOR : MHSE
FAMILY : Conveyor
VERSION : 3.0
// ATTRIBUTES
// AUTO_NUMBER = True
// BLOCK_NUMBER = 219
// END_ATTRIBUTES
   VAR_INPUT
      ix_PEC { ExternalAccessible := 'False'; ExternalVisible := 'False'; ExternalWritable := 'False'} : Bool;   // Signal of the PEC
      iUDT_PECConfiguration { ExternalAccessible := 'False'; ExternalVisible := 'False'; ExternalWritable := 'False'} : "UDT_PECConfiguration";   // PEC configuration structure
   END_VAR

   VAR_OUTPUT
      qx_PECFiltered { ExternalAccessible := 'False'; ExternalVisible := 'False'; ExternalWritable := 'False'} : Bool;   // PEC Filtered
      qUDT_HMIStatus { ExternalAccessible := 'False'; ExternalVisible := 'False'; ExternalWritable := 'False'} : "UDT_PECStatus";   // Status structure
   END_VAR

   VAR_IN_OUT
      iqUDT_ConveyorInterface : "UDT_ConveyorInterface";   // Interface structure
      iqUDT_PECStatistics : "UDT_PECStatistics";   // Statistics structure
   END_VAR

   VAR
      s_Status { ExternalAccessible := 'False'; ExternalVisible := 'False'; ExternalWritable := 'False'; S7_SetPoint := 'False'} : "UDT_PECStatus";   // Status structure
      s_StatusOld { ExternalAccessible := 'False'; ExternalVisible := 'False'; ExternalWritable := 'False'; S7_SetPoint := 'False'} : "UDT_PECStatus";   // Auxiliary status structure
      sx_Enable { ExternalAccessible := 'False'; ExternalVisible := 'False'; ExternalWritable := 'False'} : Bool;   // Enable
   END_VAR
   VAR RETAIN
      si_AuxJamDisplacement { ExternalAccessible := 'False'; ExternalVisible := 'False'; ExternalWritable := 'False'} : Int;   // Auxiliary variable to calculate displacement when PEC is blocked
   END_VAR
   VAR
      sx_PECFiltered { ExternalAccessible := 'False'; ExternalVisible := 'False'; ExternalWritable := 'False'} : Bool;   // Photo eye filtered
      PEC_TimerOnOffDelay { ExternalAccessible := 'False'; ExternalVisible := 'False'; ExternalWritable := 'False'; S7_SetPoint := 'False'} : "FB_TimerOnOffDelay";   // Filtering end of section photo eye signal
      R_TRIG_PECJam {InstructionName := 'R_TRIG'; LibVersion := '1.0'; ExternalAccessible := 'False'; ExternalVisible := 'False'; ExternalWritable := 'False'; S7_SetPoint := 'False'} : R_TRIG;   // Rising edge trigger PEC jam
   END_VAR


BEGIN
	(*
	----------------------------------------------------------------------------------------

	Version history:
	Date        | Version   | Author        | Remark
	----------------------------------------------------------------------------------------
	04/10/2019  | 2.0       | S. Nikodem    | first release TIA 15.1
	09/10/2019  | 2.1       | L.Klar        | Internal PEC error added
	28/10/2019  | 2.2       | S. Nikodem    | Change sign in region 2 - equal to greater then
	29/10/2019  | 2.3       | L.Klar        | UDT_PECStatus output variable changed, interface comments adjusted
	29/10/2019  | 2.4       | L.Klar        | Region 4 - time input corrected
	12/11/2019  | 3.0       | P.Majka       | 3.0 MHS library release TIA 15.1
	26/11/2019  | 3.1       | P.Majka       | Static variable name change to PEC from EOS PEC
	12/12/2019  | 3.2       | C. Leite      | Absolute displacement value to control jam error in both directions
	21/02/2023  | 4.0       | F.Baten       | 4.0 Release TIA 17.5
	12/03/2024  | 4.1       | S. Nieswiec   | Small variable name changes according to current standard
	*)

	REGION 1 - Triggers

	    // Rising edge PEC Jam
	    #R_TRIG_PECJam(CLK := #s_Status.Jam);

	END_REGION

	REGION 2 - Active function

	    // To activate the jam monitoring the jam displacement limit  must be configured up to zero.
	    #sx_Enable := #iUDT_PECConfiguration.JamDisplacementLimit > 0;

	END_REGION

	REGION 3 - Reset errors

	    // Jam error is reset when reset bit is active and jam error is active and is connfigured alllow reset jam with PEC blocked or photo eye is not active
	    IF #iqUDT_ConveyorInterface.InternalErrorReset
	        AND (#iUDT_PECConfiguration.ResetWithPECBlocked
	        OR (NOT #iUDT_PECConfiguration.ResetWithPECBlocked
	        AND #sx_PECFiltered))
	        AND #s_Status.Jam
	    THEN

	        #si_AuxJamDisplacement := 0;
	        #s_Status.Jam := FALSE;

	    END_IF;

	END_REGION

	REGION 4 - Photo eye filters

	    // End of section photo eye signal filter timer
	    #PEC_TimerOnOffDelay(iudi_OnDelayTime := #iUDT_PECConfiguration.TimeOnDelay,
	                         iudi_OffDelayTime := #iUDT_PECConfiguration.TimeOffDelay,
	                         ix_SignalToDelay := #ix_PEC,
	                         ix_Enable := TRUE,
	                         qx_DelayedSignal => #sx_PECFiltered);

	    // Write the current status of the photo eye
	    #s_Status.PEC := #sx_PECFiltered;
	    #qx_PECFiltered := #sx_PECFiltered;

	END_REGION

	REGION 5 - Jam detection

	    IF NOT #sx_PECFiltered                                                    // Photo eye blocked
	        AND #sx_Enable                                                            // Active of checking the PEC jam
	    THEN

	        #si_AuxJamDisplacement += ABS(#iqUDT_ConveyorInterface.Displacement);

	    ELSE

	        #si_AuxJamDisplacement := 0;

	    END_IF;

	    // Compare jam auxiliary counter with displacement jam configured
	    IF #si_AuxJamDisplacement > #iUDT_PECConfiguration.JamDisplacementLimit
	    THEN

	        #s_Status.Jam := TRUE;

	    END_IF;

	END_REGION

	REGION 6 - Statistics

	    // Statistics Jam PEC
	    IF #s_Status.Jam                                                                // PEC jam error active
	        OR #iqUDT_ConveyorInterface.ResetStatistics                                       // Reset statistics
	    THEN

	        "FC_Statistics"(ix_Reset := #iqUDT_ConveyorInterface.ResetStatistics,
	                        ix_Activate := #s_Status.Jam,
	                        ix_RTrigActivate := #R_TRIG_PECJam.Q,
	                        iqUDT_Statistics := #iqUDT_PECStatistics.Jam);

	    END_IF;

	END_REGION

	REGION 7 - Internal PEC error

	    IF #s_Status.Jam
	    THEN

	        #iqUDT_ConveyorInterface.InternalErrorPEC := TRUE;

	    END_IF;

	END_REGION


	REGION 8 - Status

	    // Status update on change
	    IF #s_StatusOld <> #s_Status
	    THEN

	        #qUDT_HMIStatus := #s_Status;
	        #s_StatusOld := #s_Status;

	    END_IF;

	END_REGION
END_FUNCTION_BLOCK

FUNCTION "FC_TimeToString" : Void
TITLE = FC_TimeToString
{ S7_Optimized_Access := 'TRUE' }
AUTHOR : MHSE
FAMILY : GeneralSystemFunctions
VERSION : 3.0
// ATTRIBUTES
// AUTO_NUMBER = True
// BLOCK_NUMBER = 29
// END_ATTRIBUTES
//Function to convert date in DTL to the string format.
   VAR_INPUT
      ia_Date {InstructionName := 'DTL'; LibVersion := '1.0'} : DTL;   // DTL format date
   END_VAR

   VAR_OUTPUT
      qs_Date : String;   // String format date
   END_VAR

   VAR_TEMP
      ta_StringDate : Struct   // String format date
         Year : String;   //   Year
         Month : String[2];   //   Month
         Day : String[2];   //   Day
         Hour : String[2];   //   Hour
         Minute : String[2];   //   Minunte
         Second : String[2];   //   Second
         Millisecond : String[4];   //   Millisecond
      END_STRUCT;
      ta_HTAReturn : Struct   // HTA operation status
         Year : Word;   //   Year
         Month : Word;   //   Month
         Day : Word;   //   Day
         Hour : Word;   //   Hour
         Minute : Word;   //   Minunte
         Second : Word;   //   Second
         Millisecond : Word;   //   Millisecond
      END_STRUCT;
   END_VAR

   VAR CONSTANT
      ci_Positions4 : USInt := 4;   // Number of character positions
      ci_DecimalPlaces0 : USInt := 0;   // Number of decimal places
      ci_Format0 : USInt := 0;   // Output format of the characters
      ci_Position1 : USInt := 1;   // Character starting at which the result is written
      cc_Colon : Char := ':';   // Colon sign
   END_VAR


BEGIN
	(*
	----------------------------------------------------------------------------------------

	Version history:
	Date        | Version   | Author        | Remark
	----------------------------------------------------------------------------------------
	24/05/2019  | 0.1       | K.Pokorski    | first release MHS TIA 15.1
	24/07/2019  | 2.0       | L.Klar        | 2.0 MHS library release TIA 15.1
	27/08/2019  | 2.1       | M.Kurpiers    | Comments adjusted
	05/09/2019  | 2.2       | K.Pokorski    | FC changed from unoptimized to optimized
	12/11/2019  | 3.0       | P.Majka       | 3.0 MHS library release TIA 15.1
	16/02/2023  | 3.1       | F.Baten       | Added constants
	21/02/2023  | 4.0       | F.Baten       | 4.0 Release TIA 17.5
	*)

	REGION 1 - Date and time separation

	    // Convert the year into a character string
	    VAL_STRG(IN := #ia_Date.YEAR,
	             SIZE := #ci_Positions4,
	             PREC := #ci_DecimalPlaces0,
	             FORMAT := USINT_TO_WORD(#ci_Format0),
	             P := #ci_Position1,
	             OUT => #ta_StringDate.Year);

	    // Using the HTA function, convert date into a string format
	    #ta_HTAReturn.Month := HTA(IN := WORD_TO_BYTE(INT_TO_BCD16((USINT_TO_INT(#ia_Date.MONTH)))), N := 1, OUT => #ta_StringDate.Month);                          // Convert the month
	    #ta_HTAReturn.Day := HTA(IN := WORD_TO_BYTE(INT_TO_BCD16((USINT_TO_INT(#ia_Date.DAY)))), N := 1, OUT => #ta_StringDate.Day);                                // Convert the day
	    #ta_HTAReturn.Hour := HTA(IN := WORD_TO_BYTE(INT_TO_BCD16((USINT_TO_INT(#ia_Date.HOUR)))), N := 1, OUT => #ta_StringDate.Hour);                             // Convert the hour
	    #ta_HTAReturn.Minute := HTA(IN := WORD_TO_BYTE(INT_TO_BCD16((USINT_TO_INT(#ia_Date.MINUTE)))), N := 1, OUT => #ta_StringDate.Minute);                       // Convert the minute
	    #ta_HTAReturn.Second := HTA(IN := WORD_TO_BYTE(INT_TO_BCD16((USINT_TO_INT(#ia_Date.SECOND)))), N := 1, OUT => #ta_StringDate.Second);                       // Convert the second
	    #ta_HTAReturn.Millisecond := HTA(IN := INT_TO_BCD16((UDINT_TO_INT(#ia_Date.NANOSECOND / 1000000))), N := 2, OUT => #ta_StringDate.Millisecond);              // Convert the millisecond

	END_REGION

	REGION 2 - Timestamp preparation

	    // Combine several input strings into one long output string
	    #qs_Date := (CONCAT(IN1 := #ta_StringDate.Year,
	                        IN2 := #cc_Colon,
	                        IN3 := #ta_StringDate.Month,
	                        IN4 := #cc_Colon,
	                        IN5 := #ta_StringDate.Day,
	                        IN6 := #cc_Colon,
	                        IN7 := #ta_StringDate.Hour,
	                        IN8 := #cc_Colon,
	                        IN9 := #ta_StringDate.Minute,
	                        IN10 := #cc_Colon,
	                        IN11 := #ta_StringDate.Second,
	                        IN12 := #cc_Colon,
	                        IN13 := RIGHT(IN := #ta_StringDate.Millisecond, L := 3)));

	END_REGION
END_FUNCTION

FUNCTION_BLOCK "FB_EncoderFault"
TITLE = Block to handle encoder fault , statistics
{ S7_Optimized_Access := 'TRUE' }
VERSION : 0.1
// ATTRIBUTES
// AUTO_NUMBER = True
// BLOCK_NUMBER = 8
// END_ATTRIBUTES
   VAR_INPUT
      ix_EncoderPulses { ExternalAccessible := 'False'; ExternalVisible := 'False'; ExternalWritable := 'False'} : Bool;   // Signal from encoder
   END_VAR

   VAR_OUTPUT
      qUDT_HMIStatus { ExternalAccessible := 'False'; ExternalVisible := 'False'; ExternalWritable := 'False'} : "UDT_EncoderStatus";   // Encoder fault status
   END_VAR

